KUKA KRL program: MyProgram_141().src

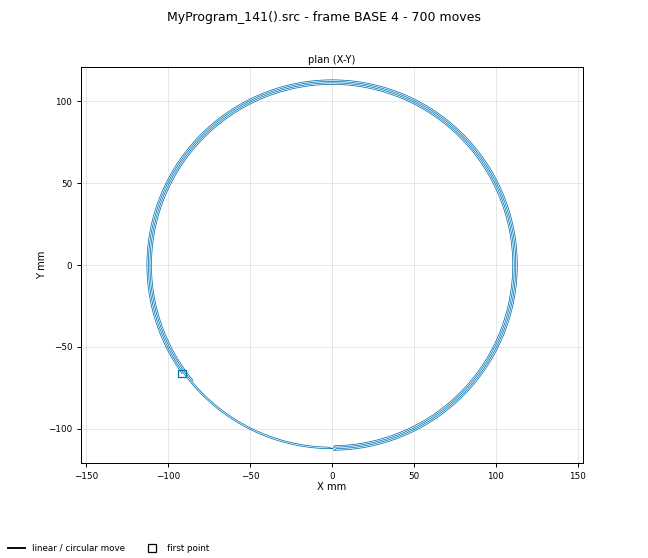
[picture p0: tool path of MyProgram_141().src in frame BASE 4, 700 of 700 moves have a stored position in this frame; points joined in program order, loops and branches not executed]
&ACCESS RVP
&REL 1
&PARAM TEMPLATE = C:\KRC\Roboter\Template\vorgabe
&PARAM EDITMASK = *
DEF MyProgram_141()
; ---- Setting reference (Base) ----
$BASE = BASE_DATA[4]

; --------------------------
; ---- Setting tool (TCP) ----
$TOOL = TOOL_DATA[3]
; --------------------------

$VEL.CP = VEL_APROX_PRINT
Startdeposition()
$VEL.CP = VEL_PRINT
LIN {X -91.6624,Y -66.2535,Z 113,A -148.3007,B 24.9515,C -1.6085,E1 24.8697,E2 234.2722} C_DIS
LIN {X -93.2607,Y -63.984,Z 113,A -149.7147,B 24.9513,C -1.6118,E1 24.8675,E2 235.6855} C_DIS
LIN {X -95.2768,Y -60.9377,Z 113,A -151.5758,B 24.9511,C -1.6162,E1 24.8646,E2 237.5454} C_DIS
LIN {X -96.7436,Y -58.5812,Z 113,A -152.9901,B 24.9508,C -1.6196,E1 24.8626,E2 238.9588} C_DIS
LIN {X -98.1521,Y -56.1893,Z 113,A -154.4681,B 24.9508,C -1.6206,E1 24.8605,E2 240.4422} C_DIS
LIN {X -99.7449,Y -53.3148,Z 113,A -156.2521,B 24.9508,C -1.6204,E1 24.8581,E2 242.2361} C_DIS
LIN {X -101.3464,Y -50.1991,Z 113,A -157.8945,B 24.9502,C -1.6306,E1 24.8561,E2 243.863} C_DIS
LIN {X -102.8265,Y -47.098,Z 113,A -159.6163,B 24.9498,C -1.6363,E1 24.854,E2 245.5806} C_DIS
LIN {X -103.9236,Y -44.624,Z 113,A -160.981,B 24.9496,C -1.6405,E1 24.8525,E2 246.9428} C_DIS
LIN {X -105.5211,Y -40.704,Z 113,A -163.1541,B 24.9493,C -1.6456,E1 24.8502,E2 249.1158} C_DIS
LIN {X -106.7787,Y -37.2743,Z 113,A -165.0805,B 24.9491,C -1.6482,E1 24.8484,E2 251.047} C_DIS
LIN {X -108.1071,Y -33.2262,Z 113,A -167.1751,B 24.9485,C -1.6572,E1 24.8466,E2 253.1321} C_DIS
LIN {X -108.8635,Y -30.6564,Z 113,A -168.6194,B 24.9485,C -1.658,E1 24.8455,E2 254.583} C_DIS
LIN {X -109.9181,Y -26.6287,Z 113,A -170.6791,B 24.948,C -1.6664,E1 24.8441,E2 256.6346} C_DIS
LIN {X -110.6473,Y -23.4242,Z 113,A -172.3554,B 24.9477,C -1.6711,E1 24.8431,E2 258.3095} C_DIS
LIN {X -111.3441,Y -19.8383,Z 113,A -174.2824,B 24.9475,C -1.674,E1 24.8421,E2 260.241} C_DIS
LIN {X -111.7974,Y -17.0998,Z 113,A -175.6982,B 24.9472,C -1.6781,E1 24.8415,E2 261.6556} C_DIS
LIN {X -112.3511,Y -12.9732,Z 113,A -177.8222,B 24.9468,C -1.6842,E1 24.8407,E2 263.7775} C_DIS
LIN {X -112.6356,Y -10.2121,Z 113,A -179.2383,B 24.9466,C -1.6884,E1 24.8403,E2 265.1923} C_DIS
LIN {X -112.8868,Y -6.9354,Z 113,A 179.149,B 24.9461,C -1.6957,E1 24.84,E2 266.7972} C_DIS
LIN {X -113.001,Y -4.673,Z 113,A 177.9295,B 24.9461,C -1.6967,E1 24.8399,E2 268.0217} C_DIS
LIN {X -113.097,Y -0.5539,Z 113,A 175.7974,B 24.9457,C -1.7017,E1 24.8398,E2 270.1548} C_DIS
LIN {X -113.0655,Y 2.7756,Z 113,A 174.1926,B 24.9452,C -1.7103,E1 24.8398,E2 271.7486} C_DIS
LIN {X -112.9676,Y 5.4512,Z 113,A 172.8457,B 24.9449,C -1.7151,E1 24.84,E2 273.0923} C_DIS
LIN {X -112.8276,Y 7.8107,Z 113,A 171.6206,B 24.9447,C -1.7179,E1 24.8402,E2 274.3179} C_DIS
LIN {X -112.555,Y 11.0857,Z 113,A 169.944,B 24.9444,C -1.7228,E1 24.8407,E2 275.9929} C_DIS
LIN {X -112.249,Y 13.8446,Z 113,A 168.5279,B 24.9441,C -1.727,E1 24.8411,E2 277.4075} C_DIS
LIN {X -111.9473,Y 16.0896,Z 113,A 167.3084,B 24.9441,C -1.728,E1 24.8416,E2 278.6319} C_DIS
LIN {X -111.4345,Y 19.3357,Z 113,A 165.6956,B 24.9436,C -1.7354,E1 24.8423,E2 280.2368} C_DIS
LIN {X -110.75,Y 22.924,Z 113,A 163.8317,B 24.9432,C -1.7408,E1 24.8433,E2 282.0987} C_DIS
LIN {X -110.0391,Y 26.1326,Z 113,A 162.1555,B 24.9429,C -1.7457,E1 24.8444,E2 283.7731} C_DIS
LIN {X -109.3647,Y 28.8252,Z 113,A 160.7396,B 24.9426,C -1.7498,E1 24.8453,E2 285.1874} C_DIS
LIN {X -108.3748,Y 32.3415,Z 113,A 158.8759,B 24.9423,C -1.7552,E1 24.8468,E2 287.0491} C_DIS
LIN {X -107.5485,Y 34.9914,Z 113,A 157.4602,B 24.942,C -1.7593,E1 24.848,E2 288.4632} C_DIS
LIN {X -106.4883,Y 38.1021,Z 113,A 155.7838,B 24.9417,C -1.764,E1 24.8495,E2 290.1378} C_DIS
LIN {X -105.2004,Y 41.5206,Z 113,A 153.857,B 24.9415,C -1.7668,E1 24.8514,E2 292.0687} C_DIS
LIN {X -103.6008,Y 45.3645,Z 113,A 151.7972,B 24.9409,C -1.7752,E1 24.8537,E2 294.12} C_DIS
LIN {X -102.2408,Y 48.3563,Z 113,A 150.1215,B 24.9406,C -1.7798,E1 24.8556,E2 295.794} C_DIS
LIN {X -100.6241,Y 51.6321,Z 113,A 148.1949,B 24.9405,C -1.7824,E1 24.8581,E2 297.7247} C_DIS
LIN {X -99.0832,Y 54.5348,Z 113,A 146.5831,B 24.94,C -1.7893,E1 24.8602,E2 299.3284} C_DIS
LIN {X -97.9694,Y 56.5073,Z 113,A 145.3647,B 24.94,C -1.7899,E1 24.8619,E2 300.5518} C_DIS
LIN {X -96.5531,Y 58.8945,Z 113,A 143.9497,B 24.9397,C -1.7936,E1 24.8639,E2 301.9652} C_DIS
LIN {X -94.8029,Y 61.676,Z 113,A 142.3381,B 24.9392,C -1.8004,E1 24.8663,E2 303.5688} C_DIS
LIN {X -92.4685,Y 65.1237,Z 113,A 140.2161,B 24.9389,C -1.8058,E1 24.8697,E2 305.6885} C_DIS
LIN {X -90.8425,Y 67.3734,Z 113,A 138.8015,B 24.9386,C -1.8093,E1 24.872,E2 307.1016} C_DIS
LIN {X -88.6177,Y 70.2707,Z 113,A 136.9398,B 24.9383,C -1.8139,E1 24.8752,E2 308.9611} C_DIS
LIN {X -86.5401,Y 72.8171,Z 113,A 135.2656,B 24.9381,C -1.8179,E1 24.8782,E2 310.6337} C_DIS
LIN {X -84.1419,Y 75.5726,Z 113,A 133.4046,B 24.9378,C -1.8222,E1 24.8816,E2 312.4926} C_DIS
LIN {X -81.9121,Y 77.9868,Z 113,A 131.7306,B 24.9375,C -1.826,E1 24.8848,E2 314.165} C_DIS
LIN {X -79.9735,Y 79.9735,Z 113,A 130.317,B 24.9373,C -1.8292,E1 24.8875,E2 315.5771} C_DIS
LIN {X -77.3477,Y 82.5131,Z 113,A 128.4565,B 24.937,C -1.8332,E1 24.8913,E2 317.4356} C_DIS
LIN {X -75.2994,Y 84.3864,Z 113,A 127.0431,B 24.9368,C -1.8362,E1 24.8942,E2 318.8476} C_DIS
LIN {X -73.2058,Y 86.209,Z 113,A 125.6303,B 24.9366,C -1.8391,E1 24.8972,E2 320.2589} C_DIS
LIN {X -71.0681,Y 87.9796,Z 113,A 124.217,B 24.9364,C -1.8419,E1 24.9003,E2 321.6708} C_DIS
LIN {X -68.4831,Y 90.0088,Z 113,A 122.5445,B 24.9362,C -1.8452,E1 24.9039,E2 323.3419} C_DIS
LIN {X -65.1237,Y 92.4685,Z 113,A 120.4259,B 24.9359,C -1.8491,E1 24.9087,E2 325.4583} C_DIS
LIN {X -62.1023,Y 94.5218,Z 113,A 118.5671,B 24.9357,C -1.8525,E1 24.913,E2 327.3154} C_DIS
LIN {X -59.764,Y 96.0174,Z 113,A 117.155,B 24.9355,C -1.8549,E1 24.9164,E2 328.7261} C_DIS
LIN {X -57.5917,Y 97.3357,Z 113,A 115.8128,B 24.9355,C -1.8551,E1 24.9196,E2 330.0721} C_DIS
LIN {X -55.0035,Y 98.8214,Z 113,A 114.2756,B 24.9354,C -1.8567,E1 24.9233,E2 331.6098} C_DIS
LIN {X -52.0867,Y 100.3917,Z 113,A 112.6607,B 24.935,C -1.8621,E1 24.9273,E2 333.2165} C_DIS
LIN {X -50.0648,Y 101.4129,Z 113,A 111.4638,B 24.935,C -1.862,E1 24.9303,E2 334.4168} C_DIS
LIN {X -47.098,Y 102.8265,Z 113,A 109.8386,B 24.9347,C -1.8661,E1 24.9344,E2 336.0362} C_DIS
LIN {X -44.5603,Y 103.9514,Z 113,A 108.4276,B 24.9346,C -1.868,E1 24.938,E2 337.4461} C_DIS
LIN {X -42.0475,Y 104.9926,Z 113,A 107.0448,B 24.9345,C -1.8698,E1 24.9416,E2 338.8278} C_DIS
LIN {X -39.406,Y 106.0127,Z 113,A 105.6067,B 24.9343,C -1.8715,E1 24.9453,E2 340.2648} C_DIS
LIN {X -35.83,Y 107.2723,Z 113,A 103.6446,B 24.9343,C -1.8723,E1 24.9505,E2 342.229} C_DIS
LIN {X -32.8311,Y 108.2296,Z 113,A 102.0821,B 24.9341,C -1.8754,E1 24.9547,E2 343.7867} C_DIS
LIN {X -28.8252,Y 109.3647,Z 113,A 99.968,B 24.9339,C -1.8774,E1 24.9604,E2 345.8993} C_DIS
LIN {X -25.2778,Y 110.2366,Z 113,A 98.0502,B 24.9339,C -1.8764,E1 24.9656,E2 347.822} C_DIS
LIN {X -22.5648,Y 110.8237,Z 113,A 96.6414,B 24.9339,C -1.8775,E1 24.9694,E2 349.2299} C_DIS
LIN {X -19.8383,Y 111.3441,Z 113,A 95.2326,B 24.9339,C -1.8785,E1 24.9733,E2 350.6378} C_DIS
LIN {X -17.0998,Y 111.7974,Z 113,A 93.8243,B 24.9338,C -1.8794,E1 24.9772,E2 352.0453} C_DIS
LIN {X -13.8446,Y 112.249,Z 113,A 92.2208,B 24.9335,C -1.883,E1 24.9816,E2 353.6416} C_DIS
LIN {X -11.0857,Y 112.555,Z 113,A 90.8126,B 24.9335,C -1.8836,E1 24.9855,E2 355.049} C_DIS
LIN {X -7.8107,Y 112.8276,Z 113,A 89.1098,B 24.9335,C -1.8828,E1 24.9902,E2 356.7544} C_DIS
LIN {X -4.673,Y 113.001,Z 113,A 87.4895,B 24.9335,C -1.8822,E1 24.9948,E2 358.3766} C_DIS
LIN {X -1.8984,Y 113.0817,Z 113,A 86.0825,B 24.9335,C -1.8825,E1 24.9987,E2 359.7829} C_DIS
LIN {X 0.8773,Y 113.0942,Z 113,A 84.6757,B 24.9335,C -1.8828,E1 25.0026,E2 361.189} C_DIS
LIN {X 3.6525,Y 113.0386,Z 113,A 83.2692,B 24.9335,C -1.8829,E1 25.0066,E2 362.595} C_DIS
LIN {X 7.8107,Y 112.8276,Z 113,A 81.1598,B 24.9335,C -1.8829,E1 25.0124,E2 364.7035} C_DIS
LIN {X 11.0857,Y 112.555,Z 113,A 79.5585,B 24.9334,C -1.8854,E1 25.0169,E2 366.2981} C_DIS
LIN {X 13.8446,Y 112.249,Z 113,A 78.1528,B 24.9334,C -1.8852,E1 25.0208,E2 367.7033} C_DIS
LIN {X 17.9668,Y 111.6634,Z 113,A 76.0447,B 24.9334,C -1.8846,E1 25.0266,E2 369.8107} C_DIS
LIN {X 20.7017,Y 111.1888,Z 113,A 74.6394,B 24.9334,C -1.8841,E1 25.0304,E2 371.2156} C_DIS
LIN {X 24.2814,Y 110.4603,Z 113,A 72.7275,B 24.9337,C -1.8807,E1 25.0357,E2 373.1332} C_DIS
LIN {X 28.3307,Y 109.4918,Z 113,A 70.6209,B 24.9337,C -1.8796,E1 25.0414,E2 375.2394} C_DIS
LIN {X 32.3415,Y 108.3748,Z 113,A 68.5776,B 24.9337,C -1.8809,E1 25.0469,E2 377.2761} C_DIS
LIN {X 35.4773,Y 107.3913,Z 113,A 66.9158,B 24.9337,C -1.8797,E1 25.0513,E2 378.9378} C_DIS
LIN {X 38.1021,Y 106.4883,Z 113,A 65.5124,B 24.9338,C -1.8785,E1 25.055,E2 380.3411} C_DIS
LIN {X 41.5206,Y 105.2004,Z 113,A 63.6021,B 24.9342,C -1.8742,E1 25.06,E2 382.2574} C_DIS
LIN {X 45.3646,Y 103.6008,Z 113,A 61.5608,B 24.9342,C -1.8749,E1 25.0652,E2 384.2924} C_DIS
LIN {X 47.8934,Y 102.4563,Z 113,A 60.1581,B 24.9342,C -1.8734,E1 25.0688,E2 385.695} C_DIS
LIN {X 50.4481,Y 101.223,Z 113,A 58.6745,B 24.9345,C -1.8695,E1 25.0725,E2 387.1838} C_DIS
LIN {X 53.3148,Y 99.7449,Z 113,A 57.0957,B 24.9345,C -1.8697,E1 25.0764,E2 388.7577} C_DIS
LIN {X 55.7466,Y 98.4065,Z 113,A 55.6935,B 24.9345,C -1.8679,E1 25.0798,E2 390.1601} C_DIS
LIN {X 58.8945,Y 96.5531,Z 113,A 53.8489,B 24.9348,C -1.8655,E1 25.0842,E2 392.0047} C_DIS
LIN {X 61.2463,Y 95.0787,Z 113,A 52.3843,B 24.9351,C -1.8607,E1 25.0877,E2 393.476} C_DIS
LIN {X 63.984,Y 93.2607,Z 113,A 50.7882,B 24.9351,C -1.8609,E1 25.0914,E2 395.0661} C_DIS
LIN {X 66.7663,Y 91.2869,Z 113,A 49.0153,B 24.9354,C -1.856,E1 25.0954,E2 396.8444} C_DIS
LIN {X 69.5825,Y 89.1617,Z 113,A 47.2861,B 24.9354,C -1.8553,E1 25.0992,E2 398.569} C_DIS
LIN {X 71.7496,Y 87.4272,Z 113,A 45.8855,B 24.9356,C -1.8529,E1 25.1023,E2 399.97} C_DIS
LIN {X 74.5344,Y 85.0629,Z 113,A 44.0427,B 24.9359,C -1.8496,E1 25.1062,E2 401.8133} C_DIS
LIN {X 76.9757,Y 82.8629,Z 113,A 42.385,B 24.9361,C -1.8465,E1 25.1096,E2 403.4716} C_DIS
LIN {X 78.782,Y 81.1456,Z 113,A 41.1061,B 24.9363,C -1.8432,E1 25.1122,E2 404.7532} C_DIS
LIN {X 80.9489,Y 78.9861,Z 113,A 39.5855,B 24.9365,C -1.8411,E1 25.1152,E2 406.2722} C_DIS
LIN {X 83.456,Y 76.3293,Z 113,A 37.7435,B 24.9367,C -1.8374,E1 25.1187,E2 408.1149} C_DIS
LIN {X 85.2305,Y 74.3424,Z 113,A 36.3792,B 24.937,C -1.8336,E1 25.1212,E2 409.4819} C_DIS
LIN {X 87.1008,Y 72.1424,Z 113,A 34.9452,B 24.9371,C -1.8315,E1 25.1238,E2 410.9144} C_DIS
LIN {X 88.8451,Y 69.9831,Z 113,A 33.4832,B 24.9375,C -1.8256,E1 25.1263,E2 412.3835} C_DIS
LIN {X 91.3607,Y 66.6655,Z 113,A 31.4479,B 24.9377,C -1.8237,E1 25.1297,E2 414.4136} C_DIS
LIN {X 92.9693,Y 64.4033,Z 113,A 29.9866,B 24.9381,C -1.8176,E1 25.1321,E2 415.8821} C_DIS
LIN {X 95.2768,Y 60.9377,Z 113,A 27.8889,B 24.9384,C -1.8127,E1 25.1353,E2 417.981} C_DIS
LIN {X 97.0088,Y 58.1448,Z 113,A 26.2963,B 24.9384,C -1.8114,E1 25.1376,E2 419.5683} C_DIS
LIN {X 98.8342,Y 54.9806,Z 113,A 24.4069,B 24.939,C -1.8047,E1 25.1402,E2 421.4638} C_DIS
LIN {X 100.1537,Y 52.5385,Z 113,A 22.9957,B 24.9392,C -1.8006,E1 25.1421,E2 422.8774} C_DIS
LIN {X 101.8609,Y 49.1471,Z 113,A 21.1008,B 24.9395,C -1.7964,E1 25.1444,E2 424.7718} C_DIS
LIN {X 103.187,Y 46.2982,Z 113,A 19.5015,B 24.9398,C -1.7915,E1 25.1463,E2 426.3741} C_DIS
LIN {X 104.4904,Y 43.2813,Z 113,A 17.91,B 24.9399,C -1.79,E1 25.148,E2 427.9605} C_DIS
LIN {X 106.0127,Y 39.406,Z 113,A 15.8138,B 24.9403,C -1.7844,E1 25.1501,E2 430.0583} C_DIS
LIN {X 107.2281,Y 35.9611,Z 113,A 13.9748,B 24.9407,C -1.7794,E1 25.1518,E2 431.8987} C_DIS
LIN {X 108.2296,Y 32.8311,Z 113,A 12.3208,B 24.941,C -1.7748,E1 25.1532,E2 433.5542} C_DIS
LIN {X 109.3647,Y 28.8252,Z 113,A 10.2255,B 24.9414,C -1.7689,E1 25.1548,E2 435.6513} C_DIS
LIN {X 110.0391,Y 26.1326,Z 113,A 8.8283,B 24.9416,C -1.765,E1 25.1557,E2 437.0497} C_DIS
LIN {X 110.6473,Y 23.4242,Z 113,A 7.4316,B 24.9419,C -1.761,E1 25.1565,E2 438.4476} C_DIS
LIN {X 111.3441,Y 19.8383,Z 113,A 5.5934,B 24.9422,C -1.7558,E1 25.1575,E2 440.2874} C_DIS
LIN {X 111.7974,Y 17.0998,Z 113,A 4.1339,B 24.9427,C -1.7489,E1 25.1581,E2 441.7546} C_DIS
LIN {X 112.249,Y 13.8446,Z 113,A 2.5434,B 24.9428,C -1.7469,E1 25.1587,E2 443.3403} C_DIS
LIN {X 112.555,Y 11.0857,Z 113,A 1.1463,B 24.9431,C -1.7428,E1 25.1591,E2 444.7387} C_DIS
LIN {X 112.8868,Y 6.9353,Z 113,A -0.9482,B 24.9435,C -1.7367,E1 25.1595,E2 446.8353} C_DIS
LIN {X 113.001,Y 4.673,Z 113,A -2.1507,B 24.9439,C -1.7305,E1 25.1597,E2 448.0453} C_DIS
LIN {X 113.097,Y 0.5539,Z 113,A -4.2532,B 24.9444,C -1.723,E1 25.1597,E2 450.1529} C_DIS
LIN {X 113.0655,Y -2.7756,Z 113,A -5.8358,B 24.9444,C -1.7223,E1 25.1597,E2 451.7278} C_DIS
LIN {X 112.9149,Y -6.4255,Z 113,A -7.6739,B 24.9448,C -1.7169,E1 25.1595,E2 453.5678} C_DIS
LIN {X 112.7232,Y -9.1946,Z 113,A -9.1329,B 24.9452,C -1.7099,E1 25.1592,E2 455.0346} C_DIS
LIN {X 112.4637,Y -11.9582,Z 113,A -10.5296,B 24.9455,C -1.7057,E1 25.1588,E2 456.4328} C_DIS
LIN {X 112.0707,Y -15.221,Z 113,A -12.12,B 24.9456,C -1.7037,E1 25.1582,E2 458.0186} C_DIS
LIN {X 111.6634,Y -17.9668,Z 113,A -13.5164,B 24.9459,C -1.6996,E1 25.1576,E2 459.4165} C_DIS
LIN {X 111.1888,Y -20.7017,Z 113,A -14.913,B 24.9461,C -1.6955,E1 25.1569,E2 460.8146} C_DIS
LIN {X 110.6473,Y -23.4242,Z 113,A -16.3098,B 24.9464,C -1.6914,E1 25.1561,E2 462.2129} C_DIS
LIN {X 109.7102,Y -27.481,Z 113,A -18.4043,B 24.9468,C -1.6853,E1 25.1548,E2 464.3097} C_DIS
LIN {X 108.6249,Y -31.4982,Z 113,A -20.498,B 24.9472,C -1.6792,E1 25.1532,E2 466.4057} C_DIS
LIN {X 107.5485,Y -34.9914,Z 113,A -22.3374,B 24.9475,C -1.674,E1 25.1517,E2 468.247} C_DIS
LIN {X 106.4883,Y -38.1021,Z 113,A -23.9911,B 24.9478,C -1.6692,E1 25.1502,E2 469.9026} C_DIS
LIN {X 105.2004,Y -41.5206,Z 113,A -25.8926,B 24.9483,C -1.6611,E1 25.1483,E2 471.8125} C_DIS
LIN {X 103.9514,Y -44.5603,Z 113,A -27.4836,B 24.9484,C -1.6594,E1 25.1466,E2 473.399} C_DIS
LIN {X 102.8265,Y -47.098,Z 113,A -28.8805,B 24.9486,C -1.6555,E1 25.1449,E2 474.7974} C_DIS
LIN {X 101.6397,Y -49.6073,Z 113,A -30.2777,B 24.9489,C -1.6516,E1 25.1433,E2 476.1961} C_DIS
LIN {X 100.6241,Y -51.6321,Z 113,A -31.4181,B 24.9491,C -1.6486,E1 25.1418,E2 477.3378} C_DIS
LIN {X 99.3267,Y -54.0859,Z 113,A -32.8155,B 24.9493,C -1.6448,E1 25.14,E2 478.7367} C_DIS
LIN {X 97.715,Y -56.95,Z 113,A -34.4698,B 24.9496,C -1.6403,E1 25.1377,E2 480.393} C_DIS
LIN {X 96.2879,Y -59.3309,Z 113,A -35.8672,B 24.9498,C -1.6367,E1 25.1356,E2 481.7918} C_DIS
LIN {X 94.8029,Y -61.676,Z 113,A -37.265,B 24.95,C -1.633,E1 25.1335,E2 483.1912} C_DIS
LIN {X 93.2607,Y -63.984,Z 113,A -38.663,B 24.9502,C -1.6295,E1 25.1313,E2 484.5907} C_DIS
LIN {X 91.1441,Y -66.9614,Z 113,A -40.5026,B 24.9505,C -1.6249,E1 25.1283,E2 486.4323} C_DIS
LIN {X 89.4733,Y -69.178,Z 113,A -41.9632,B 24.9509,C -1.6186,E1 25.1259,E2 487.9009} C_DIS
LIN {X 87.4272,Y -71.7496,Z 113,A -43.556,B 24.9509,C -1.6174,E1 25.1231,E2 489.489} C_DIS
LIN {X 85.64,Y -73.8736,Z 113,A -44.9545,B 24.9512,C -1.614,E1 25.1205,E2 490.889} C_DIS
LIN {X 83.2081,Y -76.5995,Z 113,A -46.7951,B 24.9514,C -1.6098,E1 25.1171,E2 492.7315} C_DIS
LIN {X 81.3032,Y -78.6184,Z 113,A -48.2563,B 24.9518,C -1.6037,E1 25.1143,E2 494.2007} C_DIS
LIN {X 79.3494,Y -80.59,Z 113,A -49.6553,B 24.952,C -1.6006,E1 25.1115,E2 495.601} C_DIS
LIN {X 76.9757,Y -82.8629,Z 113,A -51.2485,B 24.952,C -1.5998,E1 25.1083,E2 497.1896} C_DIS
LIN {X 74.919,Y -84.727,Z 113,A -52.6478,B 24.9522,C -1.5968,E1 25.1053,E2 498.5903} C_DIS
LIN {X 72.1424,Y -87.1008,Z 113,A -54.4897,B 24.9524,C -1.5931,E1 25.1014,E2 500.434} C_DIS
LIN {X 69.9831,Y -88.845,Z 113,A -55.952,B 24.9528,C -1.5874,E1 25.0982,E2 501.9041} C_DIS
LIN {X 67.3734,Y -90.8425,Z 113,A -57.5464,B 24.9528,C -1.587,E1 25.0947,E2 503.4938} C_DIS
LIN {X 65.1237,Y -92.4685,Z 113,A -58.9464,B 24.953,C -1.5844,E1 25.0915,E2 504.8952} C_DIS
LIN {X 62.1023,Y -94.5218,Z 113,A -60.7893,B 24.9532,C -1.581,E1 25.0872,E2 506.7397} C_DIS
LIN {X 59.764,Y -96.0174,Z 113,A -62.1897,B 24.9533,C -1.5786,E1 25.0839,E2 508.1414} C_DIS
LIN {X 57.3896,Y -97.4552,Z 113,A -63.5903,B 24.9534,C -1.5762,E1 25.0805,E2 509.5433} C_DIS
LIN {X 54.5348,Y -99.0832,Z 113,A -65.2489,B 24.9536,C -1.5735,E1 25.0765,E2 511.2035} C_DIS
LIN {X 52.0867,Y -100.3917,Z 113,A -66.6498,B 24.9537,C -1.5713,E1 25.073,E2 512.6056} C_DIS
LIN {X 48.8166,Y -102.0197,Z 113,A -68.557,B 24.9541,C -1.5658,E1 25.0682,E2 514.5208} C_DIS
LIN {X 46.2982,Y -103.187,Z 113,A -69.9586,B 24.9541,C -1.5638,E1 25.0647,E2 515.9235} C_DIS
LIN {X 42.4688,Y -104.8212,Z 113,A -72.0612,B 24.9543,C -1.561,E1 25.0592,E2 518.0278} C_DIS
LIN {X 39.406,Y -106.0127,Z 113,A -73.6585,B 24.9543,C -1.5617,E1 25.0551,E2 519.6201} C_DIS
LIN {X 35.4773,Y -107.3913,Z 113,A -75.7619,B 24.9544,C -1.5592,E1 25.0495,E2 521.7251} C_DIS
LIN {X 32.8311,Y -108.2296,Z 113,A -77.1646,B 24.9545,C -1.5577,E1 25.0458,E2 523.1288} C_DIS
LIN {X 28.8252,Y -109.3647,Z 113,A -79.269,B 24.9547,C -1.5556,E1 25.0401,E2 525.2348} C_DIS
LIN {X 25.2778,Y -110.2366,Z 113,A -81.1787,B 24.9549,C -1.5513,E1 25.0349,E2 527.1521} C_DIS
LIN {X 21.2032,Y -111.0923,Z 113,A -83.2213,B 24.9549,C -1.5523,E1 25.0293,E2 529.1896} C_DIS
LIN {X 17.9668,Y -111.6634,Z 113,A -84.8834,B 24.9549,C -1.5511,E1 25.0248,E2 530.8528} C_DIS
LIN {X 15.221,Y -112.0707,Z 113,A -86.2875,B 24.9549,C -1.5502,E1 25.0209,E2 532.2577} C_DIS
LIN {X 11.0857,Y -112.555,Z 113,A -88.3944,B 24.955,C -1.5491,E1 25.015,E2 534.3659} C_DIS
LIN {X 8.3201,Y -112.7932,Z 113,A -89.7987,B 24.955,C -1.5485,E1 25.0111,E2 535.7709} C_DIS
LIN {X 5.5495,Y -112.9634,Z 113,A -91.2041,B 24.9551,C -1.548,E1 25.0072,E2 537.1771} C_DIS
LIN {X 2.9206,Y -113.0611,Z 113,A -92.5119,B 24.9551,C -1.5486,E1 25.0035,E2 538.4831} C_DIS
LIN {X 0.7926,Y -113.0921,Z 113,A -93.1683,B 24.954,C -1.5666,E1 25.0018,E2 539.0966} C_DIS
Enddeposition()
LIN {X 0.7926,Y -113.0921,Z 113,A -93.1683,B 24.954,C -1.5666,E1 25.0018,E2 539.0966} C_DIS
Startdeposition()
$VEL.CP = VEL_PRINT
LIN {X 2.5112,Y -112.1455,Z 113,A -92.1451,B 24.9527,C -1.5891,E1 25.0049,E2 538.0202} C_DIS
LIN {X 8.5342,Y -111.8483,Z 113,A -89.0646,B 24.9527,C -1.5904,E1 25.0134,E2 534.938} C_DIS
LIN {X 11.7323,Y -111.5575,Z 113,A -87.3874,B 24.9525,C -1.5929,E1 25.0181,E2 533.2559} C_DIS
LIN {X 14.4396,Y -111.2394,Z 113,A -85.9602,B 24.9523,C -1.5953,E1 25.0221,E2 531.8241} C_DIS
LIN {X 17.4758,Y -110.8035,Z 113,A -84.3472,B 24.9521,C -1.5984,E1 25.0265,E2 530.2052} C_DIS
LIN {X 20.9501,Y -110.1992,Z 113,A -82.5997,B 24.9521,C -1.5975,E1 25.0313,E2 528.4617} C_DIS
LIN {X 23.9582,Y -109.5843,Z 113,A -81.0272,B 24.9521,C -1.5991,E1 25.0356,E2 526.8874} C_DIS
LIN {X 27.7429,Y -108.688,Z 113,A -78.9698,B 24.9518,C -1.6042,E1 25.0412,E2 524.821} C_DIS
LIN {X 31.8742,Y -107.5488,Z 113,A -76.8637,B 24.9518,C -1.603,E1 25.0469,E2 522.7212} C_DIS
LIN {X 35.1139,Y -106.5368,Z 113,A -75.0751,B 24.9516,C -1.6075,E1 25.0516,E2 520.9253} C_DIS
LIN {X 38.3768,Y -105.4037,Z 113,A -73.3742,B 24.9516,C -1.607,E1 25.0561,E2 519.229} C_DIS
LIN {X 41.5145,Y -104.2092,Z 113,A -71.46,B 24.9509,C -1.6183,E1 25.0611,E2 517.2924} C_DIS
LIN {X 44.6783,Y -102.8911,Z 113,A -69.8639,B 24.9512,C -1.614,E1 25.0652,E2 515.7103} C_DIS
LIN {X 49.5705,Y -100.6258,Z 113,A -67.1605,B 24.9511,C -1.6162,E1 25.072,E2 513.0087} C_DIS
LIN {X 52.3888,Y -99.1874,Z 113,A -65.6255,B 24.9511,C -1.6153,E1 25.0758,E2 511.4802} C_DIS
LIN {X 55.0783,Y -97.7204,Z 113,A -63.9299,B 24.9506,C -1.6239,E1 25.08,E2 509.7691} C_DIS
LIN {X 58.6737,Y -95.6052,Z 113,A -62.0003,B 24.9509,C -1.6189,E1 25.0846,E2 507.8574} C_DIS
LIN {X 61.0092,Y -94.132,Z 113,A -60.5316,B 24.9506,C -1.6242,E1 25.088,E2 506.3808} C_DIS
LIN {X 64.0536,Y -92.0861,Z 113,A -58.5905,B 24.9501,C -1.6311,E1 25.0925,E2 504.4301} C_DIS
LIN {X 67.1129,Y -89.8815,Z 113,A -56.7131,B 24.9501,C -1.6329,E1 25.0968,E2 502.555} C_DIS
LIN {X 70.2089,Y -87.4855,Z 113,A -54.8395,B 24.9501,C -1.6316,E1 25.1009,E2 500.6916} C_DIS
LIN {X 72.6167,Y -85.4959,Z 113,A -53.0723,B 24.9494,C -1.643,E1 25.1047,E2 498.9042} C_DIS
LIN {X 75.0079,Y -83.4061,Z 113,A -51.4123,B 24.9491,C -1.6485,E1 25.1082,E2 497.2379} C_DIS
LIN {X 77.8348,Y -80.7741,Z 113,A -49.55,B 24.9491,C -1.6482,E1 25.1119,E2 495.3839} C_DIS
LIN {X 80.4847,Y -78.1351,Z 113,A -47.5426,B 24.9485,C -1.6573,E1 25.1159,E2 493.3635} C_DIS
LIN {X 83.1854,Y -75.2546,Z 113,A -45.5747,B 24.9483,C -1.6602,E1 25.1196,E2 491.3975} C_DIS
LIN {X 85.5486,Y -72.5549,Z 113,A -43.7264,B 24.948,C -1.6658,E1 25.123,E2 489.5445} C_DIS
LIN {X 88.0435,Y -69.5058,Z 113,A -41.8472,B 24.948,C -1.665,E1 25.1262,E2 487.6757} C_DIS
LIN {X 89.9009,Y -67.087,Z 113,A -40.2598,B 24.9477,C -1.6706,E1 25.1289,E2 486.0826} C_DIS
LIN {X 91.8394,Y -64.4085,Z 113,A -38.4603,B 24.9471,C -1.6804,E1 25.1319,E2 484.2688} C_DIS
LIN {X 94.7779,Y -60.0021,Z 113,A -35.8423,B 24.9469,C -1.6841,E1 25.1359,E2 481.6553} C_DIS
LIN {X 96.7147,Y -56.8248,Z 113,A -34.0662,B 24.9469,C -1.6839,E1 25.1384,E2 479.8887} C_DIS
LIN {X 98.2445,Y -54.1399,Z 113,A -32.4123,B 24.9464,C -1.692,E1 25.1407,E2 478.2243} C_DIS
LIN {X 100.6478,Y -49.5261,Z 113,A -30.158,B 24.947,C -1.6814,E1 25.1435,E2 476.0068} C_DIS
LIN {X 101.7078,Y -47.31,Z 113,A -28.5242,B 24.9457,C -1.7027,E1 25.1455,E2 474.3319} C_DIS
LIN {X 103.5972,Y -43.0195,Z 113,A -26.2509,B 24.9456,C -1.7044,E1 25.148,E2 472.0669} C_DIS
LIN {X 104.7364,Y -40.1649,Z 113,A -24.5203,B 24.9448,C -1.7167,E1 25.1498,E2 470.3169} C_DIS
LIN {X 105.9424,Y -36.8647,Z 113,A -22.9043,B 24.9449,C -1.7141,E1 25.1513,E2 468.716} C_DIS
LIN {X 106.9636,Y -33.791,Z 113,A -21.167,B 24.9444,C -1.7231,E1 25.1528,E2 466.9673} C_DIS
LIN {X 107.9761,Y -30.3958,Z 113,A -19.4367,B 24.9442,C -1.7252,E1 25.1541,E2 465.2419} C_DIS
LIN {X 108.853,Y -27.0925,Z 113,A -17.7976,B 24.9442,C -1.7259,E1 25.1553,E2 463.6107} C_DIS
LIN {X 109.5657,Y -24.0433,Z 113,A -16.0317,B 24.9433,C -1.7387,E1 25.1564,E2 461.8248} C_DIS
LIN {X 110.3068,Y -20.3814,Z 113,A -14.1646,B 24.9431,C -1.743,E1 25.1574,E2 459.9586} C_DIS
LIN {X 110.8378,Y -17.254,Z 113,A -12.4625,B 24.9425,C -1.752,E1 25.1581,E2 458.2451} C_DIS
LIN {X 111.3567,Y -13.5133,Z 113,A -10.1714,B 24.9409,C -1.7751,E1 25.1589,E2 455.9132} C_DIS
LIN {X 111.7451,Y -9.7981,Z 113,A -8.8111,B 24.9422,C -1.7559,E1 25.1593,E2 454.6062} C_DIS
LIN {X 112.062,Y -4.9855,Z 113,A -6.6068,B 24.9425,C -1.752,E1 25.1597,E2 452.4243} C_DIS
LIN {X 112.1495,Y -2.2913,Z 113,A -4.9394,B 24.9413,C -1.7698,E1 25.1597,E2 450.7247} C_DIS
LIN {X 112.1668,Y 1.309,Z 113,A -2.9928,B 24.9406,C -1.7808,E1 25.1597,E2 448.7639} C_DIS
LIN {X 112.0632,Y 4.9571,Z 113,A -1.224,B 24.9405,C -1.7824,E1 25.1596,E2 447.0017} C_DIS
LIN {X 111.8321,Y 8.7368,Z 113,A 0.6673,B 24.9402,C -1.7867,E1 25.1592,E2 445.1116} C_DIS
LIN {X 111.5367,Y 11.9304,Z 113,A 2.2567,B 24.94,C -1.7897,E1 25.1588,E2 443.5245} C_DIS
LIN {X 111.0858,Y 15.5789,Z 113,A 4.1552,B 24.9395,C -1.7966,E1 25.1581,E2 441.6208} C_DIS
LIN {X 110.5476,Y 19.0322,Z 113,A 6.027,B 24.9388,C -1.8063,E1 25.1572,E2 439.7373} C_DIS
LIN {X 109.8105,Y 22.9015,Z 113,A 7.8832,B 24.9389,C -1.8054,E1 25.1562,E2 437.8938} C_DIS
LIN {X 109.027,Y 26.3793,Z 113,A 9.7018,B 24.9385,C -1.811,E1 25.1551,E2 436.0727} C_DIS
LIN {X 108.1044,Y 29.9431,Z 113,A 11.8899,B 24.9372,C -1.8309,E1 25.1534,E2 433.8501} C_DIS
LIN {X 106.752,Y 34.449,Z 113,A 14.0135,B 24.9375,C -1.8254,E1 25.1517,E2 431.7517} C_DIS
LIN {X 105.6578,Y 37.6756,Z 113,A 15.8302,B 24.9369,C -1.8341,E1 25.15,E2 429.9247} C_DIS
LIN {X 103.8793,Y 42.3298,Z 113,A 18.1635,B 24.9371,C -1.832,E1 25.1477,E2 427.6094} C_DIS
LIN {X 102.5513,Y 45.4579,Z 113,A 20.1472,B 24.936,C -1.8483,E1 25.1454,E2 425.598} C_DIS
LIN {X 101.1808,Y 48.4271,Z 113,A 21.6412,B 24.9362,C -1.845,E1 25.1436,E2 424.1198} C_DIS
LIN {X 99.6449,Y 51.5159,Z 113,A 23.4735,B 24.9356,C -1.8531,E1 25.1413,E2 422.2782} C_DIS
LIN {X 97.8767,Y 54.7985,Z 113,A 25.2621,B 24.9356,C -1.8531,E1 25.1389,E2 420.499} C_DIS
LIN {X 95.8357,Y 58.2943,Z 113,A 27.2678,B 24.9354,C -1.8558,E1 25.1361,E2 418.4971} C_DIS
LIN {X 94.1883,Y 60.9215,Z 113,A 28.9898,B 24.9347,C -1.8662,E1 25.1335,E2 416.7591} C_DIS
LIN {X 91.8164,Y 64.4416,Z 113,A 31.1083,B 24.9345,C -1.8695,E1 25.1301,E2 414.6433} C_DIS
LIN {X 89.8392,Y 67.1691,Z 113,A 33.2028,B 24.933,C -1.8908,E1 25.1266,E2 412.5087} C_DIS
LIN {X 87.6788,Y 69.9664,Z 113,A 34.4506,B 24.9345,C -1.8699,E1 25.1245,E2 411.316} C_DIS
LIN {X 86.2115,Y 71.7655,Z 113,A 35.7535,B 24.9339,C -1.878,E1 25.1222,E2 409.9999} C_DIS
LIN {X 84.3142,Y 73.9857,Z 113,A 38.4395,B 24.9298,C -1.9356,E1 25.117,E2 407.19} C_DIS
LIN {X 79.6225,Y 79.0129,Z 113,A 40.65,B 24.9334,C -1.8843,E1 25.1129,E2 405.11} C_DIS
LIN {X 77.1108,Y 81.4663,Z 113,A 42.5453,B 24.9328,C -1.8927,E1 25.1091,E2 403.203} C_DIS
LIN {X 74.6437,Y 83.7322,Z 113,A 44.2075,B 24.9328,C -1.894,E1 25.1056,E2 401.5444} C_DIS
LIN {X 72.224,Y 85.8305,Z 113,A 46.1022,B 24.9317,C -1.9086,E1 25.1015,E2 399.6224} C_DIS
LIN {X 69.3952,Y 88.1309,Z 113,A 47.7592,B 24.9321,C -1.903,E1 25.098,E2 397.9849} C_DIS
LIN {X 66.5837,Y 90.2744,Z 113,A 49.4846,B 24.9321,C -1.9027,E1 25.0941,E2 396.2665} C_DIS
LIN {X 63.8801,Y 92.2067,Z 113,A 51.1892,B 24.9319,C -1.9059,E1 25.0902,E2 394.5602} C_DIS
LIN {X 60.4321,Y 94.5025,Z 113,A 53.3724,B 24.9314,C -1.9122,E1 25.0851,E2 392.3691} C_DIS
LIN {X 56.9256,Y 96.6552,Z 113,A 55.4975,B 24.9311,C -1.9164,E1 25.08,E2 390.2407} C_DIS
LIN {X 53.5657,Y 98.5568,Z 113,A 57.419,B 24.9311,C -1.917,E1 25.0753,E2 388.3235} C_DIS
LIN {X 50.218,Y 100.3049,Z 113,A 59.3265,B 24.931,C -1.9185,E1 25.0706,E2 386.4176} C_DIS
LIN {X 47.1976,Y 101.7601,Z 113,A 60.9948,B 24.931,C -1.9187,E1 25.0664,E2 384.7533} C_DIS
LIN {X 44.5978,Y 102.9263,Z 113,A 62.4366,B 24.931,C -1.9197,E1 25.0627,E2 383.3125} C_DIS
LIN {X 39.7619,Y 104.889,Z 113,A 65.0881,B 24.9308,C -1.9218,E1 25.0558,E2 380.6621} C_DIS
LIN {X 36.9792,Y 105.9022,Z 113,A 66.5834,B 24.9308,C -1.9224,E1 25.0519,E2 379.1683} C_DIS
LIN {X 33.7832,Y 106.9661,Z 113,A 68.5526,B 24.9298,C -1.9345,E1 25.0466,E2 377.1741} C_DIS
LIN {X 28.9249,Y 108.3798,Z 113,A 70.8823,B 24.9305,C -1.9253,E1 25.0404,E2 374.8701} C_DIS
LIN {X 26.5374,Y 108.9884,Z 113,A 72.2083,B 24.9302,C -1.929,E1 25.0368,E2 373.5375} C_DIS
LIN {X 22.4898,Y 109.8951,Z 113,A 74.2886,B 24.9302,C -1.9284,E1 25.0311,E2 371.4612} C_DIS
LIN {X 18.8205,Y 110.583,Z 113,A 76.2275,B 24.9302,C -1.9304,E1 25.0258,E2 369.5196} C_DIS
LIN {X 15.4258,Y 111.1075,Z 113,A 78.0589,B 24.9299,C -1.9342,E1 25.0207,E2 367.6809} C_DIS
LIN {X 11.6901,Y 111.5619,Z 113,A 79.838,B 24.9303,C -1.9284,E1 25.0158,E2 365.9167} C_DIS
LIN {X 8.5342,Y 111.8483,Z 113,A 81.6027,B 24.9298,C -1.9347,E1 25.0109,E2 364.138} C_DIS
LIN {X 4.6784,Y 112.0752,Z 113,A 83.4431,B 24.9302,C -1.9291,E1 25.0058,E2 362.3116} C_DIS
LIN {X 0.9332,Y 112.1691,Z 113,A 85.4241,B 24.93,C -1.9316,E1 25.0002,E2 360.3249} C_DIS
LIN {X -2.5688,Y 112.1444,Z 113,A 87.0799,B 24.9305,C -1.9256,E1 24.9956,E2 358.6832} C_DIS
LIN {X -5.2848,Y 112.0491,Z 113,A 88.6698,B 24.9299,C -1.9336,E1 24.9911,E2 357.0741} C_DIS
LIN {X -9.527,Y 111.7689,Z 113,A 90.8489,B 24.9299,C -1.933,E1 24.9851,E2 354.8955} C_DIS
LIN {X -13.1388,Y 111.4006,Z 113,A 92.5474,B 24.9305,C -1.9255,E1 24.9804,E2 353.2138} C_DIS
LIN {X -16.3964,Y 110.9696,Z 113,A 94.4753,B 24.9298,C -1.9347,E1 24.975,E2 351.2623} C_DIS
LIN {X -20.6054,Y 110.2655,Z 113,A 96.5241,B 24.9303,C -1.9276,E1 24.9694,E2 349.2284} C_DIS
LIN {X -23.8315,Y 109.6119,Z 113,A 98.0937,B 24.9308,C -1.9216,E1 24.9652,E2 347.6712} C_DIS
LIN {X -26.9861,Y 108.879,Z 113,A 99.936,B 24.9303,C -1.9278,E1 24.9601,E2 345.8117} C_DIS
LIN {X -31.2506,Y 107.7338,Z 113,A 102.6543,B 24.9291,C -1.9445,E1 24.9527,E2 343.0494} C_DIS
LIN {X -35.2766,Y 106.483,Z 113,A 104.2874,B 24.9309,C -1.9204,E1 24.9485,E2 341.4704} C_DIS
LIN {X -38.5104,Y 105.3549,Z 113,A 105.9824,B 24.9312,C -1.916,E1 24.9441,E2 339.7825} C_DIS
LIN {X -43.4392,Y 103.4203,Z 113,A 108.3547,B 24.9324,C -1.8987,E1 24.938,E2 337.4461} C_DIS
LIN {X -47.0891,Y 101.8106,Z 113,A 110.7629,B 24.9316,C -1.9107,E1 24.9318,E2 335.0037} C_DIS
LIN {X -51.1534,Y 99.8301,Z 113,A 112.6323,B 24.9331,C -1.8892,E1 24.9272,E2 333.1805} C_DIS
LIN {X -54.4111,Y 98.0931,Z 113,A 115.0157,B 24.9319,C -1.906,E1 24.9213,E2 330.7504} C_DIS
LIN {X -57.967,Y 96.0347,Z 113,A 117.4555,B 24.9312,C -1.916,E1 24.9153,E2 328.2794} C_DIS
LIN {X -60.8822,Y 94.2135,Z 113,A 118.7279,B 24.9328,C -1.8931,E1 24.9124,E2 327.0574} C_DIS
LIN {X -63.4968,Y 92.4731,Z 113,A 120.4695,B 24.9327,C -1.8954,E1 24.9084,E2 325.3045} C_DIS
LIN {X -66.4364,Y 90.3823,Z 113,A 122.2479,B 24.9331,C -1.8891,E1 24.9044,E2 323.5349} C_DIS
LIN {X -69.5533,Y 88.006,Z 113,A 124.2045,B 24.9335,C -1.883,E1 24.9001,E2 321.5857} C_DIS
LIN {X -71.7345,Y 86.2373,Z 113,A 125.766,B 24.9334,C -1.8849,E1 24.8967,E2 320.0137} C_DIS
LIN {X -74.3359,Y 84.0075,Z 113,A 127.595,B 24.9334,C -1.884,E1 24.8928,E2 318.1796} C_DIS
LIN {X -77.2426,Y 81.3424,Z 113,A 129.6857,B 24.9336,C -1.8823,E1 24.8886,E2 316.0844} C_DIS
LIN {X -80.1311,Y 78.498,Z 113,A 131.6917,B 24.9341,C -1.8747,E1 24.8846,E2 314.0881} C_DIS
LIN {X -82.6374,Y 75.8536,Z 113,A 133.4468,B 24.9347,C -1.8658,E1 24.8813,E2 312.3464} C_DIS
LIN {X -85.1716,Y 72.9974,Z 113,A 135.589,B 24.9346,C -1.8684,E1 24.8774,E2 310.1884} C_DIS
LIN {X -89.245,Y 67.9592,Z 113,A 138.672,B 24.9358,C -1.8506,E1 24.8721,E2 307.1333} C_DIS
LIN {X -91.132,Y 65.4046,Z 113,A 140.4009,B 24.9358,C -1.8504,E1 24.8692,E2 305.3965} C_DIS
LIN {X -93.2596,Y 62.3362,Z 113,A 142.8955,B 24.9346,C -1.8683,E1 24.8652,E2 302.8468} C_DIS
LIN {X -95.5337,Y 58.7913,Z 113,A 144.3651,B 24.9369,C -1.8352,E1 24.8632,E2 301.4486} C_DIS
LIN {X -97.4592,Y 55.539,Z 113,A 146.427,B 24.9369,C -1.8348,E1 24.8602,E2 299.3771} C_DIS
LIN {X -99.2698,Y 52.2323,Z 113,A 148.3864,B 24.9372,C -1.8304,E1 24.8577,E2 297.4177} C_DIS
LIN {X -101.0156,Y 48.7709,Z 113,A 150.3696,B 24.9376,C -1.8246,E1 24.8552,E2 295.4376} C_DIS
LIN {X -102.4191,Y 45.7512,Z 113,A 152.1982,B 24.9376,C -1.8244,E1 24.8531,E2 293.5994} C_DIS
LIN {X -104.1692,Y 41.6159,Z 113,A 154.2678,B 24.9387,C -1.8086,E1 24.8509,E2 291.556} C_DIS
LIN {X -104.9992,Y 39.4709,Z 113,A 155.6301,B 24.9384,C -1.8123,E1 24.8495,E2 290.1773} C_DIS
LIN {X -106.1419,Y 36.2883,Z 113,A 158.023,B 24.937,C -1.8331,E1 24.8474,E2 287.7212} C_DIS
LIN {X -107.5997,Y 31.7026,Z 113,A 159.6337,B 24.9398,C -1.792,E1 24.8461,E2 286.1991} C_DIS
LIN {X -108.827,Y 27.1991,Z 113,A 162.0691,B 24.9402,C -1.7864,E1 24.8444,E2 283.763} C_DIS
LIN {X -109.5471,Y 24.1286,Z 113,A 163.7872,B 24.9402,C -1.7854,E1 24.8433,E2 282.0371} C_DIS
LIN {X -110.3529,Y 20.125,Z 113,A 165.6165,B 24.9414,C -1.7687,E1 24.8423,E2 280.2368} C_DIS
LIN {X -110.6972,Y 18.1374,Z 113,A 166.9357,B 24.9408,C -1.7766,E1 24.8417,E2 278.8909} C_DIS
LIN {X -111.2782,Y 14.1406,Z 113,A 168.949,B 24.9414,C -1.768,E1 24.8409,E2 276.8862} C_DIS
LIN {X -111.6561,Y 10.7624,Z 113,A 170.731,B 24.9417,C -1.7641,E1 24.8404,E2 275.1027} C_DIS
LIN {X -111.9636,Y 6.8803,Z 113,A 172.6769,B 24.9422,C -1.7559,E1 24.84,E2 273.1646} C_DIS
LIN {X -112.1101,Y 3.7604,Z 113,A 174.3004,B 24.9425,C -1.7519,E1 24.8398,E2 271.541} C_DIS
LIN {X -112.1725,Y 0.4893,Z 113,A 176.0039,B 24.9428,C -1.7477,E1 24.8398,E2 269.8371} C_DIS
LIN {X -112.1381,Y -2.8475,Z 113,A 177.7433,B 24.943,C -1.7436,E1 24.8398,E2 268.0972} C_DIS
LIN {X -112.0431,Y -5.4255,Z 113,A 179.1559,B 24.943,C -1.743,E1 24.8401,E2 266.6774} C_DIS
LIN {X -111.8272,Y -8.7986,Z 113,A -179.2143,B 24.9437,C -1.7337,E1 24.8404,E2 265.06} C_DIS
LIN {X -111.5594,Y -11.7139,Z 113,A -177.6566,B 24.9438,C -1.7314,E1 24.8408,E2 263.4986} C_DIS
LIN {X -111.1052,Y -15.4421,Z 113,A -175.818,B 24.9444,C -1.7221,E1 24.8415,E2 261.671} C_DIS
LIN {X -110.6796,Y -18.2428,Z 113,A -174.2032,B 24.9443,C -1.7241,E1 24.8422,E2 260.0419} C_DIS
LIN {X -109.9208,Y -22.3645,Z 113,A -172.061,B 24.9447,C -1.7174,E1 24.8433,E2 257.9029} C_DIS
LIN {X -108.8384,Y -27.1523,Z 113,A -169.5648,B 24.9453,C -1.7092,E1 24.8449,E2 255.4118} C_DIS
LIN {X -107.909,Y -30.6327,Z 113,A -167.553,B 24.9452,C -1.7103,E1 24.8464,E2 253.3855} C_DIS
LIN {X -106.6951,Y -34.6248,Z 113,A -165.6045,B 24.9461,C -1.6967,E1 24.848,E2 251.4585} C_DIS
LIN {X -105.4255,Y -38.3169,Z 113,A -163.6145,B 24.9464,C -1.6905,E1 24.8499,E2 249.4717} C_DIS
LIN {X -104.2608,Y -41.3831,Z 113,A -161.8046,B 24.9464,C -1.6909,E1 24.8517,E2 247.6507} C_DIS
LIN {X -102.7596,Y -44.9801,Z 113,A -159.3671,B 24.9457,C -1.703,E1 24.8545,E2 245.1711} C_DIS
LIN {X -101.0872,Y -48.6219,Z 113,A -157.8376,B 24.9473,C -1.6765,E1 24.8563,E2 243.6963} C_DIS
LIN {X -98.7944,Y -53.1276,Z 113,A -155.4572,B 24.9483,C -1.6613,E1 24.8593,E2 241.3394} C_DIS
LIN {X -96.9363,Y -56.4489,Z 113,A -153.2657,B 24.948,C -1.6659,E1 24.8623,E2 239.1256} C_DIS
LIN {X -94.6629,Y -60.182,Z 113,A -151.2176,B 24.9488,C -1.6526,E1 24.8653,E2 237.0986} C_DIS
LIN {X -92.2269,Y -63.851,Z 113,A -148.8292,B 24.9488,C -1.6524,E1 24.869,E2 234.6988} C_DIS
LIN {X -90.2863,Y -66.5675,Z 113,A -146.9132,B 24.9486,C -1.6566,E1 24.8722,E2 232.7636} C_DIS
LIN {X -87.9031,Y -69.6835,Z 113,A -145.0633,B 24.9493,C -1.6456,E1 24.8754,E2 230.9312} C_DIS
LIN {X -85.6854,Y -72.3943,Z 113,A -143.1854,B 24.9493,C -1.6449,E1 24.8787,E2 229.0462} C_DIS
LIN {X -83.1623,Y -75.2803,Z 113,A -141.2928,B 24.9497,C -1.6378,E1 24.8822,E2 227.162} C_DIS
LIN {X -80.5824,Y -78.0337,Z 113,A -139.3275,B 24.9499,C -1.6351,E1 24.886,E2 225.1946} C_DIS
LIN {X -77.7577,Y -80.8484,Z 113,A -137.236,B 24.95,C -1.6331,E1 24.8902,E2 223.0992} C_DIS
LIN {X -74.8316,Y -83.564,Z 113,A -135.2763,B 24.9505,C -1.6257,E1 24.8942,E2 221.1491} C_DIS
LIN {X -72.3613,Y -85.7135,Z 113,A -133.45,B 24.9503,C -1.6287,E1 24.8981,E2 219.3085} C_DIS
LIN {X -69.8926,Y -87.7378,Z 113,A -131.8976,B 24.9507,C -1.6225,E1 24.9015,E2 217.7651} C_DIS
LIN {X -67.1402,Y -89.8609,Z 113,A -130.081,B 24.9507,C -1.621,E1 24.9055,E2 215.9455} C_DIS
LIN {X -63.882,Y -92.2054,Z 113,A -128.154,B 24.9513,C -1.6125,E1 24.9099,E2 214.0322} C_DIS
LIN {X -61.292,Y -93.9484,Z 113,A -126.2727,B 24.9507,C -1.6218,E1 24.9144,E2 212.1227} C_DIS
LIN {X -57.2981,Y -96.435,Z 113,A -124.1045,B 24.9515,C -1.6085,E1 24.9195,E2 209.9794} C_DIS
LIN {X -54.4535,Y -98.0693,Z 113,A -122.3937,B 24.9515,C -1.6076,E1 24.9236,E2 208.2656} C_DIS
LIN {X -50.8369,Y -99.9919,Z 113,A -120.3101,B 24.9518,C -1.6045,E1 24.9288,E2 206.1836} C_DIS
LIN {X -46.9577,Y -101.8718,Z 113,A -118.1566,B 24.952,C -1.5999,E1 24.9342,E2 204.0357} C_DIS
LIN {X -42.4361,Y -103.836,Z 113,A -115.568,B 24.952,C -1.6002,E1 24.9409,E2 201.4404} C_DIS
LIN {X -39.4576,Y -105.0042,Z 113,A -113.9807,B 24.9522,C -1.5967,E1 24.945,E2 199.8581} C_DIS
LIN {X -36.1347,Y -106.1937,Z 113,A -112.0404,B 24.952,C -1.6009,E1 24.9502,E2 197.904} C_DIS
LIN {X -33.3975,Y -107.0857,Z 113,A -110.6458,B 24.9522,C -1.5966,E1 24.9539,E2 196.5171} C_DIS
LIN {X -29.7397,Y -108.1597,Z 113,A -108.6588,B 24.9522,C -1.597,E1 24.9592,E2 194.526} C_DIS
LIN {X -26.2672,Y -109.0544,Z 113,A -106.9307,B 24.9525,C -1.5916,E1 24.9639,E2 192.8084} C_DIS
LIN {X -22.9341,Y -109.8038,Z 113,A -105.1445,B 24.9525,C -1.5925,E1 24.9687,E2 191.0177} C_DIS
LIN {X -19.7953,Y -110.4122,Z 113,A -103.5223,B 24.9525,C -1.5914,E1 24.9732,E2 189.3963} C_DIS
LIN {X -16.0488,Y -111.019,Z 113,A -101.5105,B 24.9524,C -1.594,E1 24.9788,E2 187.3765} C_DIS
LIN {X -12.0677,Y -111.5224,Z 113,A -99.4351,B 24.9524,C -1.5948,E1 24.9845,E2 185.2979} C_DIS
LIN {X -8.3411,Y -111.8637,Z 113,A -97.0546,B 24.9511,C -1.615,E1 24.9913,E2 182.8686} C_DIS
LIN {X -4.3313,Y -112.0901,Z 113,A -95.6519,B 24.9528,C -1.5872,E1 24.995,E2 181.5316} C_DIS
LIN {X 0.796,Y -112.1393,Z 113,A -93.8798,B 24.9549,C -1.5519,E1 24.9999,E2 179.843} C_DIS
Enddeposition()
LIN {X 0.796,Y -112.1393,Z 113,A -93.8798,B 24.9549,C -1.5519,E1 24.9998,E2 179.843} C_DIS
Startdeposition()
$VEL.CP = VEL_PRINT
LIN {X -2.5976,Y -111.2189,Z 113,A -95.7064,B 24.9542,C -1.5641,E1 24.9947,E2 181.6408} C_DIS
LIN {X -7.5291,Y -110.9928,Z 113,A -98.0111,B 24.9536,C -1.5739,E1 24.9884,E2 183.9228} C_DIS
LIN {X -11.1953,Y -110.6838,Z 113,A -99.973,B 24.9537,C -1.5712,E1 24.9829,E2 185.8921} C_DIS
LIN {X -14.5846,Y -110.2881,Z 113,A -101.7933,B 24.9539,C -1.5689,E1 24.9778,E2 187.7192} C_DIS
LIN {X -18.217,Y -109.7463,Z 113,A -103.5745,B 24.9536,C -1.574,E1 24.9729,E2 189.4899} C_DIS
LIN {X -21.5581,Y -109.1404,Z 113,A -105.3728,B 24.9536,C -1.5726,E1 24.968,E2 191.2934} C_DIS
LIN {X -24.9365,Y -108.4171,Z 113,A -107.1,B 24.9535,C -1.5757,E1 24.9633,E2 193.0157} C_DIS
LIN {X -28.4586,Y -107.5478,Z 113,A -108.8608,B 24.9532,C -1.5811,E1 24.9586,E2 194.7659} C_DIS
LIN {X -31.3684,Y -106.7342,Z 113,A -110.4565,B 24.9532,C -1.5806,E1 24.9543,E2 196.3656} C_DIS
LIN {X -37.0194,Y -104.908,Z 113,A -113.4191,B 24.9528,C -1.5869,E1 24.9464,E2 199.3185} C_DIS
LIN {X -41.9165,Y -103.049,Z 113,A -116.4549,B 24.9535,C -1.5757,E1 24.9385,E2 202.3875} C_DIS
LIN {X -45.6515,Y -101.4497,Z 113,A -118.3715,B 24.9529,C -1.5851,E1 24.9336,E2 204.2862} C_DIS
LIN {X -48.6812,Y -100.0327,Z 113,A -120.5338,B 24.9539,C -1.5694,E1 24.928,E2 206.4914} C_DIS
LIN {X -51.6225,Y -98.5458,Z 113,A -121.856,B 24.9528,C -1.5867,E1 24.9249,E2 207.776} C_DIS
LIN {X -54.8935,Y -96.7635,Z 113,A -123.8371,B 24.9528,C -1.5868,E1 24.92,E2 209.7626} C_DIS
LIN {X -57.5139,Y -95.2278,Z 113,A -125.4939,B 24.9529,C -1.5854,E1 24.916,E2 211.4278} C_DIS
LIN {X -61.126,Y -92.9501,Z 113,A -127.5447,B 24.9523,C -1.5948,E1 24.9112,E2 213.463} C_DIS
LIN {X -65.8102,Y -89.6946,Z 113,A -130.4778,B 24.952,C -1.6,E1 24.9045,E2 216.3939} C_DIS
LIN {X -68.7091,Y -87.4945,Z 113,A -132.1364,B 24.9513,C -1.6119,E1 24.9009,E2 218.0301} C_DIS
LIN {X -71.6784,Y -85.0804,Z 113,A -134.4216,B 24.9518,C -1.6031,E1 24.8959,E2 220.345} C_DIS
LIN {X -74.3565,Y -82.7481,Z 113,A -136.2192,B 24.9516,C -1.608,E1 24.8922,E2 222.138} C_DIS
LIN {X -77.1468,Y -80.1528,Z 113,A -138.1844,B 24.9513,C -1.6119,E1 24.8882,E2 224.1019} C_DIS
LIN {X -79.8615,Y -77.449,Z 113,A -140.1563,B 24.9511,C -1.6162,E1 24.8843,E2 226.0719} C_DIS
LIN {X -82.2204,Y -74.9403,Z 113,A -141.9823,B 24.9509,C -1.6181,E1 24.8809,E2 227.9015} C_DIS
LIN {X -84.5734,Y -72.2735,Z 113,A -143.7314,B 24.9505,C -1.6256,E1 24.8777,E2 229.6407} C_DIS
LIN {X -86.585,Y -69.8513,Z 113,A -145.4753,B 24.9505,C -1.6246,E1 24.8746,E2 231.3949} C_DIS
LIN {X -90.34,Y -64.9224,Z 113,A -148.5645,B 24.9498,C -1.6365,E1 24.8694,E2 234.4709} C_DIS
LIN {X -92.4469,Y -61.8871,Z 113,A -151.1815,B 24.9512,C -1.6137,E1 24.8652,E2 237.1551} C_DIS
LIN {X -94.8561,Y -58.1256,Z 113,A -152.8094,B 24.9492,C -1.6457,E1 24.8629,E2 238.7151} C_DIS
LIN {X -96.4936,Y -55.3631,Z 113,A -154.4962,B 24.9491,C -1.6489,E1 24.8605,E2 240.403} C_DIS
LIN {X -97.8438,Y -52.9405,Z 113,A -156.0393,B 24.9491,C -1.6484,E1 24.8585,E2 241.9555} C_DIS
LIN {X -99.6529,Y -49.451,Z 113,A -157.6818,B 24.9478,C -1.6688,E1 24.8564,E2 243.5581} C_DIS
LIN {X -101.9183,Y -44.5956,Z 113,A -160.6535,B 24.9478,C -1.6684,E1 24.853,E2 246.547} C_DIS
LIN {X -103.2738,Y -41.3643,Z 113,A -162.682,B 24.948,C -1.665,E1 24.8508,E2 248.5949} C_DIS
LIN {X -104.6058,Y -37.8654,Z 113,A -164.5851,B 24.9476,C -1.6717,E1 24.8489,E2 250.4927} C_DIS
LIN {X -105.7857,Y -34.4312,Z 113,A -166.3293,B 24.947,C -1.6822,E1 24.8474,E2 252.222} C_DIS
LIN {X -106.5049,Y -32.1416,Z 113,A -168.2214,B 24.9483,C -1.6609,E1 24.8458,E2 254.1756} C_DIS
LIN {X -107.6371,Y -28.1167,Z 113,A -170.5734,B 24.9483,C -1.6601,E1 24.8442,E2 256.5434} C_DIS
LIN {X -108.7878,Y -23.2703,Z 113,A -172.4879,B 24.9463,C -1.6927,E1 24.843,E2 258.3914} C_DIS
LIN {X -109.4618,Y -19.8553,Z 113,A -174.1355,B 24.9456,C -1.7039,E1 24.8422,E2 260.022} C_DIS
LIN {X -110.1397,Y -15.6633,Z 113,A -176.5584,B 24.9457,C -1.7018,E1 24.8412,E2 262.4642} C_DIS
LIN {X -110.6551,Y -11.4695,Z 113,A -178.5504,B 24.9448,C -1.7158,E1 24.8405,E2 264.4348} C_DIS
LIN {X -110.953,Y -8.1186,Z 113,A 179.7337,B 24.9444,C -1.722,E1 24.8401,E2 266.1464} C_DIS
LIN {X -111.1533,Y -4.5907,Z 113,A 177.6367,B 24.9447,C -1.7173,E1 24.8399,E2 268.267} C_DIS
LIN {X -111.2491,Y -0.2197,Z 113,A 175.4744,B 24.944,C -1.728,E1 24.8398,E2 270.4169} C_DIS
LIN {X -111.2131,Y 2.8416,Z 113,A 173.7833,B 24.944,C -1.7288,E1 24.8398,E2 272.1164} C_DIS
LIN {X -111.0042,Y 7.3611,Z 113,A 171.3813,B 24.9437,C -1.7337,E1 24.8403,E2 274.5211} C_DIS
LIN {X -110.615,Y 11.8532,Z 113,A 169.2332,B 24.9427,C -1.7478,E1 24.8409,E2 276.6485} C_DIS
LIN {X -110.1584,Y 15.5318,Z 113,A 167.4455,B 24.942,C -1.7586,E1 24.8415,E2 278.4211} C_DIS
LIN {X -109.517,Y 19.5482,Z 113,A 164.6378,B 24.9434,C -1.7384,E1 24.8429,E2 281.2936} C_DIS
LIN {X -108.665,Y 23.8332,Z 113,A 163.2886,B 24.9406,C -1.7797,E1 24.8436,E2 282.5522} C_DIS
LIN {X -107.0225,Y 30.3689,Z 113,A 159.4913,B 24.9407,C -1.7783,E1 24.8462,E2 286.375} C_DIS
LIN {X -105.4786,Y 35.361,Z 113,A 156.8221,B 24.9401,C -1.7876,E1 24.8485,E2 289.0373} C_DIS
LIN {X -104.6492,Y 37.7466,Z 113,A 155.17,B 24.9407,C -1.7783,E1 24.8501,E2 290.7209} C_DIS
LIN {X -102.7936,Y 42.5439,Z 113,A 152.7803,B 24.9395,C -1.7963,E1 24.8525,E2 293.081} C_DIS
LIN {X -101.2255,Y 46.149,Z 113,A 150.6997,B 24.9392,C -1.8004,E1 24.8549,E2 295.1635} C_DIS
LIN {X -99.6517,Y 49.4535,Z 113,A 148.8382,B 24.9388,C -1.807,E1 24.8571,E2 297.0193} C_DIS
LIN {X -97.8616,Y 52.9077,Z 113,A 146.8623,B 24.9383,C -1.8139,E1 24.8597,E2 298.9891} C_DIS
LIN {X -95.9718,Y 56.2642,Z 113,A 144.8596,B 24.938,C -1.819,E1 24.8625,E2 300.9902} C_DIS
LIN {X -92.0359,Y 62.4941,Z 113,A 140.9698,B 24.9375,C -1.8261,E1 24.8684,E2 304.8826} C_DIS
LIN {X -89.5805,Y 65.9658,Z 113,A 138.2528,B 24.9385,C -1.812,E1 24.8729,E2 307.6464} C_DIS
LIN {X -86.9843,Y 69.3545,Z 113,A 135.9878,B 24.9382,C -1.8154,E1 24.8769,E2 309.9141} C_DIS
LIN {X -84.132,Y 72.7885,Z 113,A 134.2988,B 24.9362,C -1.8446,E1 24.8798,E2 311.541} C_DIS
LIN {X -82.0206,Y 75.158,Z 113,A 132.9006,B 24.9353,C -1.8579,E1 24.8824,E2 312.9138} C_DIS
LIN {X -78.8332,Y 78.496,Z 113,A 129.8805,B 24.9366,C -1.839,E1 24.8884,E2 315.992} C_DIS
LIN {X -76.393,Y 80.8719,Z 113,A 128.5619,B 24.9352,C -1.8599,E1 24.891,E2 317.2662} C_DIS
LIN {X -74.2528,Y 82.8409,Z 113,A 127.0061,B 24.9351,C -1.8612,E1 24.8942,E2 318.8252} C_DIS
LIN {X -71.635,Y 85.1174,Z 113,A 125.0637,B 24.9352,C -1.8591,E1 24.8983,E2 320.78} C_DIS
LIN {X -66.3092,Y 89.3285,Z 113,A 121.5945,B 24.9346,C -1.8677,E1 24.906,E2 324.2416} C_DIS
LIN {X -60.9475,Y 93.0678,Z 113,A 118.0479,B 24.9346,C -1.8674,E1 24.9142,E2 327.8008} C_DIS
LIN {X -56.893,Y 95.6001,Z 113,A 115.8241,B 24.9337,C -1.8813,E1 24.9194,E2 329.9984} C_DIS
LIN {X -53.7196,Y 97.42,Z 113,A 113.8483,B 24.9337,C -1.881,E1 24.9242,E2 331.9807} C_DIS
LIN {X -50.8478,Y 98.9478,Z 113,A 112.4172,B 24.9328,C -1.8934,E1 24.9277,E2 333.3861} C_DIS
LIN {X -47.9507,Y 100.3837,Z 113,A 110.5296,B 24.9332,C -1.8873,E1 24.9325,E2 335.2933} C_DIS
LIN {X -44.0766,Y 102.1446,Z 113,A 107.6859,B 24.9348,C -1.8649,E1 24.94,E2 338.197} C_DIS
LIN {X -39.6411,Y 103.9459,Z 113,A 105.9982,B 24.9324,C -1.8989,E1 24.9441,E2 339.8072} C_DIS
LIN {X -37.3688,Y 104.7854,Z 113,A 103.6823,B 24.9353,C -1.8583,E1 24.9505,E2 342.2244} C_DIS
LIN {X -31.718,Y 106.6305,Z 113,A 101.6748,B 24.9321,C -1.9035,E1 24.9556,E2 344.1278} C_DIS
LIN {X -26.5799,Y 108.0262,Z 113,A 98.8861,B 24.9321,C -1.9044,E1 24.9631,E2 346.9186} C_DIS
LIN {X -23.1887,Y 108.8056,Z 113,A 97.1071,B 24.9319,C -1.9065,E1 24.968,E2 348.6949} C_DIS
LIN {X -20.2458,Y 109.3916,Z 113,A 95.2156,B 24.9328,C -1.8938,E1 24.9732,E2 350.6185} C_DIS
LIN {X -15.668,Y 110.139,Z 113,A 93.2137,B 24.9315,C -1.9111,E1 24.9787,E2 352.5811} C_DIS
LIN {X -12.5555,Y 110.5378,Z 113,A 91.4438,B 24.9319,C -1.9058,E1 24.9836,E2 354.3648} C_DIS
LIN {X -8.8077,Y 110.8987,Z 113,A 89.575,B 24.9316,C -1.9096,E1 24.9888,E2 356.2255} C_DIS
LIN {X -5.0201,Y 111.1348,Z 113,A 87.6222,B 24.9316,C -1.9104,E1 24.9942,E2 358.177} C_DIS
LIN {X -1.536,Y 111.2385,Z 113,A 85.7285,B 24.9318,C -1.9068,E1 24.9995,E2 360.0794} C_DIS
LIN {X 2.0213,Y 111.2295,Z 113,A 84.0642,B 24.9313,C -1.914,E1 25.0041,E2 361.7264} C_DIS
LIN {X 5.0945,Y 111.1316,Z 113,A 82.4004,B 24.9315,C -1.9108,E1 25.0088,E2 363.3973} C_DIS
LIN {X 8.7483,Y 110.9034,Z 113,A 80.5345,B 24.9315,C -1.9116,E1 25.014,E2 365.2606} C_DIS
LIN {X 12.47,Y 110.5478,Z 113,A 78.5541,B 24.9317,C -1.909,E1 25.0195,E2 367.2457} C_DIS
LIN {X 15.9628,Y 110.0972,Z 113,A 76.7692,B 24.9317,C -1.9098,E1 25.0244,E2 369.0273} C_DIS
LIN {X 19.7332,Y 109.4838,Z 113,A 74.8177,B 24.9317,C -1.9098,E1 25.0298,E2 370.9768} C_DIS
LIN {X 23.4925,Y 108.7393,Z 113,A 72.8803,B 24.9316,C -1.9104,E1 25.0351,E2 372.9104} C_DIS
LIN {X 26.2223,Y 108.1134,Z 113,A 71.2716,B 24.9321,C -1.9026,E1 25.0395,E2 374.5352} C_DIS
LIN {X 30.2662,Y 107.0516,Z 113,A 68.7518,B 24.9333,C -1.8859,E1 25.0464,E2 377.0905} C_DIS
LIN {X 33.9838,Y 105.9305,Z 113,A 67.469,B 24.9313,C -1.9144,E1 25.0496,E2 378.3034} C_DIS
LIN {X 39.2512,Y 104.0935,Z 113,A 64.2815,B 24.9324,C -1.8985,E1 25.0581,E2 381.5221} C_DIS
LIN {X 43.1412,Y 102.5423,Z 113,A 62.2845,B 24.9321,C -1.903,E1 25.0632,E2 383.5038} C_DIS
LIN {X 48.0509,Y 100.3356,Z 113,A 59.5257,B 24.9323,C -1.9003,E1 25.0702,E2 386.2619} C_DIS
LIN {X 50.9653,Y 98.8877,Z 113,A 57.8236,B 24.9325,C -1.8971,E1 25.0744,E2 387.9672} C_DIS
LIN {X 54.1578,Y 97.1753,Z 113,A 55.615,B 24.9338,C -1.8799,E1 25.0799,E2 390.2101} C_DIS
LIN {X 58.655,Y 94.5293,Z 113,A 53.4255,B 24.9325,C -1.8972,E1 25.0851,E2 392.3519} C_DIS
LIN {X 62.3902,Y 92.1062,Z 113,A 50.9613,B 24.9333,C -1.8861,E1 25.0909,E2 394.8341} C_DIS
LIN {X 65.5487,Y 89.8861,Z 113,A 49.0556,B 24.9333,C -1.8862,E1 25.0952,E2 396.7328} C_DIS
LIN {X 67.581,Y 88.369,Z 113,A 47.6532,B 24.9338,C -1.8797,E1 25.0983,E2 398.1456} C_DIS
LIN {X 70.4662,Y 86.0863,Z 113,A 45.7214,B 24.9341,C -1.8745,E1 25.1025,E2 400.0824} C_DIS
LIN {X 73.246,Y 83.7325,Z 113,A 43.9644,B 24.9341,C -1.876,E1 25.1062,E2 401.8289} C_DIS
LIN {X 75.8588,Y 81.3743,Z 113,A 42.0499,B 24.9346,C -1.8679,E1 25.1102,E2 403.7549} C_DIS
LIN {X 78.6833,Y 78.6477,Z 113,A 40.2158,B 24.9343,C -1.8718,E1 25.1138,E2 405.5721} C_DIS
LIN {X 81.0033,Y 76.2533,Z 113,A 37.95,B 24.9363,C -1.8441,E1 25.1183,E2 407.8936} C_DIS
LIN {X 83.5237,Y 73.4851,Z 113,A 36.4723,B 24.9352,C -1.8593,E1 25.1209,E2 409.3287} C_DIS
LIN {X 86.0985,Y 70.4515,Z 113,A 34.3022,B 24.9359,C -1.8491,E1 25.1248,E2 411.5128} C_DIS
LIN {X 89.376,Y 66.2454,Z 113,A 31.6971,B 24.9359,C -1.8486,E1 25.1292,E2 414.1068} C_DIS
LIN {X 91.4294,Y 63.3781,Z 113,A 30.0287,B 24.9359,C -1.8506,E1 25.1319,E2 415.7624} C_DIS
LIN {X 93.2648,Y 60.6482,Z 113,A 28.1528,B 24.9367,C -1.8381,E1 25.1348,E2 417.6584} C_DIS
LIN {X 94.9781,Y 57.9248,Z 113,A 26.1324,B 24.9381,C -1.8177,E1 25.1378,E2 419.7166} C_DIS
LIN {X 96.8655,Y 54.7125,Z 113,A 24.6313,B 24.9372,C -1.8309,E1 25.1399,E2 421.1788} C_DIS
LIN {X 98.5253,Y 51.6615,Z 113,A 22.927,B 24.9372,C -1.8297,E1 25.1421,E2 422.8769} C_DIS
LIN {X 100.0319,Y 48.683,Z 113,A 20.9459,B 24.9384,C -1.8132,E1 25.1446,E2 424.8864} C_DIS
LIN {X 101.8813,Y 44.6806,Z 113,A 18.8985,B 24.9381,C -1.8166,E1 25.1469,E2 426.9145} C_DIS
LIN {X 103.0756,Y 41.8512,Z 113,A 16.3816,B 24.9412,C -1.7706,E1 25.1496,E2 429.5261} C_DIS
LIN {X 105.177,Y 36.253,Z 113,A 14.3625,B 24.9387,C -1.8084,E1 25.1514,E2 431.4448} C_DIS
LIN {X 107.1975,Y 29.7515,Z 113,A 10.6431,B 24.9401,C -1.7881,E1 25.1544,E2 435.1908} C_DIS
LIN {X 108.2904,Y 25.4853,Z 113,A 8.5451,B 24.9401,C -1.7887,E1 25.1558,E2 437.2752} C_DIS
LIN {X 108.9966,Y 22.2674,Z 113,A 6.8955,B 24.9402,C -1.7856,E1 25.1568,E2 438.9228} C_DIS
LIN {X 109.6877,Y 18.5675,Z 113,A 4.9314,B 24.9407,C -1.7783,E1 25.1578,E2 440.8924} C_DIS
LIN {X 110.2692,Y 14.7304,Z 113,A 2.9402,B 24.9411,C -1.7722,E1 25.1585,E2 442.8861} C_DIS
LIN {X 110.6404,Y 11.6106,Z 113,A 1.3724,B 24.9413,C -1.7693,E1 25.159,E2 444.4516} C_DIS
LIN {X 110.9715,Y 7.8441,Z 113,A -0.5993,B 24.9418,C -1.762,E1 25.1595,E2 446.429} C_DIS
LIN {X 111.163,Y 4.3646,Z 113,A -2.4571,B 24.9424,C -1.7533,E1 25.1597,E2 448.296} C_DIS
LIN {X 111.2481,Y 0.4187,Z 113,A -4.4738,B 24.9428,C -1.7474,E1 25.1597,E2 450.3147} C_DIS
LIN {X 111.1979,Y -3.3372,Z 113,A -6.2921,B 24.9428,C -1.7464,E1 25.1597,E2 452.1245} C_DIS
LIN {X 111.0921,Y -5.8907,Z 113,A -7.6105,B 24.9431,C -1.742,E1 25.1595,E2 453.4455} C_DIS
LIN {X 110.8697,Y -9.171,Z 113,A -9.2266,B 24.9433,C -1.74,E1 25.1592,E2 455.0568} C_DIS
LIN {X 110.5152,Y -12.7485,Z 113,A -11.1129,B 24.9438,C -1.7324,E1 25.1586,E2 456.9498} C_DIS
LIN {X 110.1556,Y -15.5517,Z 113,A -12.9166,B 24.9451,C -1.712,E1 25.1579,E2 458.7909} C_DIS
LIN {X 109.6521,Y -18.7804,Z 113,A -14.2706,B 24.9445,C -1.7213,E1 25.1573,E2 460.115} C_DIS
LIN {X 108.9746,Y -22.3749,Z 113,A -16.1046,B 24.9447,C -1.7175,E1 25.1563,E2 461.9473} C_DIS
LIN {X 108.118,Y -26.2034,Z 113,A -18.3358,B 24.9457,C -1.7015,E1 25.1549,E2 464.2033} C_DIS
LIN {X 107.0888,Y -30.1351,Z 113,A -20.7034,B 24.9469,C -1.6825,E1 25.1531,E2 466.602} C_DIS
LIN {X 105.9611,Y -33.8892,Z 113,A -22.2385,B 24.946,C -1.6978,E1 25.1518,E2 468.0924} C_DIS
LIN {X 104.8225,Y -37.2631,Z 113,A -24.0691,B 24.9463,C -1.6922,E1 25.1502,E2 469.926} C_DIS
LIN {X 103.8129,Y -39.9923,Z 113,A -26.2402,B 24.9485,C -1.6574,E1 25.1479,E2 472.1669} C_DIS
LIN {X 102.0052,Y -44.3963,Z 113,A -27.9158,B 24.9468,C -1.6846,E1 25.1461,E2 473.7693} C_DIS
LIN {X 100.5647,Y -47.574,Z 113,A -29.7334,B 24.9472,C -1.6782,E1 25.144,E2 475.5921} C_DIS
LIN {X 96.6634,Y -55.0678,Z 113,A -34.6055,B 24.9495,C -1.642,E1 25.1375,E2 480.5241} C_DIS
LIN {X 94.6056,Y -58.531,Z 113,A -36.4848,B 24.9493,C -1.6447,E1 25.1348,E2 482.3873} C_DIS
LIN {X 92.8352,Y -61.3003,Z 113,A -38.1146,B 24.9494,C -1.6427,E1 25.1323,E2 484.0137} C_DIS
LIN {X 89.9684,Y -65.4363,Z 113,A -40.3781,B 24.949,C -1.6502,E1 25.1287,E2 486.2487} C_DIS
LIN {X 87.7767,Y -68.3495,Z 113,A -42.1316,B 24.949,C -1.6506,E1 25.1257,E2 487.9928} C_DIS
LIN {X 85.0238,Y -71.7449,Z 113,A -44.546,B 24.9498,C -1.6373,E1 25.1214,E2 490.4274} C_DIS
LIN {X 82.8021,Y -74.2962,Z 113,A -46.2077,B 24.9498,C -1.6364,E1 25.1183,E2 492.0838} C_DIS
LIN {X 80.1666,Y -77.1325,Z 113,A -48.2029,B 24.9501,C -1.6314,E1 25.1145,E2 494.0822} C_DIS
LIN {X 77.4903,Y -79.8217,Z 113,A -50.1785,B 24.9505,C -1.6256,E1 25.1106,E2 496.0631} C_DIS
LIN {X 75.017,Y -82.15,Z 113,A -51.9008,B 24.9507,C -1.6227,E1 25.107,E2 497.7853} C_DIS
LIN {X 72.4164,Y -84.4517,Z 113,A -53.6904,B 24.9509,C -1.6185,E1 25.1033,E2 499.5777} C_DIS
LIN {X 70.4373,Y -86.11,Z 113,A -55.558,B 24.9525,C -1.5918,E1 25.0991,E2 501.5012} C_DIS
LIN {X 67.1762,Y -88.6773,Z 113,A -57.1652,B 24.9514,C -1.6105,E1 25.0956,E2 503.0584} C_DIS
LIN {X 64.0926,Y -90.932,Z 113,A -59.1689,B 24.9517,C -1.6048,E1 25.0911,E2 505.0687} C_DIS
LIN {X 61.0489,Y -93.0009,Z 113,A -60.7691,B 24.9512,C -1.614,E1 25.0874,E2 506.6416} C_DIS
LIN {X 58.7668,Y -94.4595,Z 113,A -62.9078,B 24.9533,C -1.5788,E1 25.0822,E2 508.8568} C_DIS
LIN {X 55.241,Y -96.5638,Z 113,A -64.5223,B 24.9522,C -1.5967,E1 25.0784,E2 510.424} C_DIS
LIN {X 52.8763,Y -97.8786,Z 113,A -66.3637,B 24.9535,C -1.5748,E1 25.0738,E2 512.312} C_DIS
LIN {X 49.3868,Y -99.6847,Z 113,A -68.1506,B 24.9531,C -1.5817,E1 25.0693,E2 514.0778} C_DIS
LIN {X 44.7963,Y -101.8309,Z 113,A -70.2481,B 24.952,C -1.5999,E1 25.0641,E2 516.127} C_DIS
LIN {X 39.4291,Y -104.0261,Z 113,A -73.438,B 24.9528,C -1.5868,E1 25.0558,E2 519.3407} C_DIS
LIN {X 35.8633,Y -105.3092,Z 113,A -75.4101,B 24.953,C -1.5833,E1 25.0506,E2 521.3169} C_DIS
LIN {X 32.6159,Y -106.3599,Z 113,A -76.9866,B 24.9527,C -1.5891,E1 25.0465,E2 522.8769} C_DIS
LIN {X 28.3115,Y -107.587,Z 113,A -79.3376,B 24.953,C -1.5845,E1 25.0401,E2 525.2348} C_DIS
LIN {X 24.8978,Y -108.4261,Z 113,A -81.2353,B 24.9533,C -1.579,E1 25.0349,E2 527.1428} C_DIS
LIN {X 21.1985,Y -109.2096,Z 113,A -83.1687,B 24.9533,C -1.5779,E1 25.0296,E2 529.0764} C_DIS
LIN {X 18.0079,Y -109.7813,Z 113,A -84.9225,B 24.9536,C -1.573,E1 25.0248,E2 530.84} C_DIS
LIN {X 14.3612,Y -110.3171,Z 113,A -86.7122,B 24.9534,C -1.5764,E1 25.0199,E2 532.6203} C_DIS
LIN {X 11.1173,Y -110.692,Z 113,A -88.4437,B 24.9536,C -1.5733,E1 25.015,E2 534.3579} C_DIS
LIN {X 8.7483,Y -110.9034,Z 113,A -89.8429,B 24.9541,C -1.5653,E1 25.0111,E2 535.7752} C_DIS
LIN {X 3.8265,Y -111.1828,Z 113,A -92.2109,B 24.9537,C -1.5715,E1 25.0045,E2 538.1277} C_DIS
LIN {X 0.7977,Y -111.2251,Z 113,A -93.8194,B 24.9539,C -1.5694,E1 25.0001,E2 539.741} C_DIS
Enddeposition()
LIN {X 0.7977,Y -111.2251,Z 113,A -93.8194,B 24.9539,C -1.5694,E1 25.0001,E2 539.741} C_DIS
Startdeposition()
$VEL.CP = VEL_PRINT
LIN {X 1.5292,Y -110.3136,Z 113,A -92.549,B 24.9506,C -1.6229,E1 25.004,E2 538.344} C_DIS
LIN {X 5.3956,Y -110.1931,Z 113,A -90.1295,B 24.9495,C -1.6412,E1 25.0108,E2 535.882} C_DIS
LIN {X 8.9419,Y -109.9602,Z 113,A -88.8479,B 24.9509,C -1.618,E1 25.0142,E2 534.656} C_DIS
LIN {X 12.0541,Y -109.6641,Z 113,A -87.0402,B 24.9504,C -1.6267,E1 25.0193,E2 532.8288} C_DIS
LIN {X 15.4516,Y -109.2357,Z 113,A -85.362,B 24.9506,C -1.6236,E1 25.0239,E2 531.1593} C_DIS
LIN {X 19.2525,Y -108.6306,Z 113,A -83.3329,B 24.9504,C -1.6264,E1 25.0295,E2 529.1255} C_DIS
LIN {X 22.8496,Y -107.933,Z 113,A -81.3656,B 24.9502,C -1.6309,E1 25.0349,E2 527.1503} C_DIS
LIN {X 27.6827,Y -106.7938,Z 113,A -79.2284,B 24.9512,C -1.6144,E1 25.0406,E2 525.0551} C_DIS
LIN {X 33.7346,Y -105.0392,Z 113,A -75.9062,B 24.9508,C -1.6201,E1 25.0496,E2 521.7249} C_DIS
LIN {X 37.2119,Y -103.8598,Z 113,A -72.4301,B 24.9464,C -1.6915,E1 25.0591,E2 518.0872} C_DIS
LIN {X 43.8401,Y -101.2388,Z 113,A -70.1761,B 24.95,C -1.633,E1 25.0645,E2 515.9769} C_DIS
LIN {X 46.7308,Y -99.9373,Z 113,A -68.3881,B 24.9495,C -1.6418,E1 25.0691,E2 514.1727} C_DIS
LIN {X 53.8454,Y -96.2905,Z 113,A -64.4318,B 24.9495,C -1.6401,E1 25.0789,E2 510.2312} C_DIS
LIN {X 56.204,Y -94.9331,Z 113,A -62.5249,B 24.9481,C -1.6645,E1 25.0836,E2 508.2724} C_DIS
LIN {X 61.1837,Y -91.8043,Z 113,A -60.024,B 24.9492,C -1.646,E1 25.0893,E2 505.8235} C_DIS
LIN {X 64.2515,Y -89.6827,Z 113,A -57.8131,B 24.9482,C -1.6621,E1 25.0945,E2 503.5822} C_DIS
LIN {X 70.6684,Y -84.7184,Z 113,A -53.7699,B 24.9482,C -1.6636,E1 25.1033,E2 499.5503} C_DIS
LIN {X 73.1253,Y -82.6091,Z 113,A -51.9447,B 24.9475,C -1.6739,E1 25.1072,E2 497.7082} C_DIS
LIN {X 75.7969,Y -80.163,Z 113,A -50.0792,B 24.9473,C -1.6777,E1 25.111,E2 495.8413} C_DIS
LIN {X 78.4404,Y -77.5777,Z 113,A -48.2343,B 24.9472,C -1.679,E1 25.1146,E2 494.001} C_DIS
LIN {X 80.9594,Y -74.9466,Z 113,A -46.2969,B 24.9467,C -1.6858,E1 25.1184,E2 492.056} C_DIS
LIN {X 83.2246,Y -72.4216,Z 113,A -44.608,B 24.9467,C -1.6871,E1 25.1215,E2 490.3716} C_DIS
LIN {X 87.6,Y -67.0637,Z 113,A -41.1593,B 24.9465,C -1.6902,E1 25.1275,E2 486.9316} C_DIS
LIN {X 89.0674,Y -65.1014,Z 113,A -39.7649,B 24.9459,C -1.6992,E1 25.1298,E2 485.5228} C_DIS
LIN {X 92.6197,Y -59.9412,Z 113,A -36.2215,B 24.9445,C -1.7214,E1 25.1354,E2 481.9445} C_DIS
LIN {X 95.71,Y -54.8706,Z 113,A -33.4545,B 24.9448,C -1.716,E1 25.1393,E2 479.2044} C_DIS
LIN {X 99.0873,Y -48.5097,Z 113,A -29.9161,B 24.9447,C -1.718,E1 25.1439,E2 475.68} C_DIS
LIN {X 100.7818,Y -44.8826,Z 113,A -27.7492,B 24.944,C -1.7283,E1 25.1464,E2 473.5006} C_DIS
LIN {X 102.734,Y -40.2112,Z 113,A -24.5673,B 24.9418,C -1.7615,E1 25.1498,E2 470.2579} C_DIS
LIN {X 104.0493,Y -36.6736,Z 113,A -23.342,B 24.9436,C -1.7343,E1 25.1509,E2 469.1037} C_DIS
LIN {X 106.2014,Y -29.8745,Z 113,A -19.7324,B 24.9432,C -1.7416,E1 25.154,E2 465.4973} C_DIS
LIN {X 107.3812,Y -25.3122,Z 113,A -16.9434,B 24.9416,C -1.7649,E1 25.1559,E2 462.6696} C_DIS
LIN {X 108.1304,Y -21.8884,Z 113,A -15.1174,B 24.9412,C -1.771,E1 25.1569,E2 460.8397} C_DIS
LIN {X 109.2597,Y -15.2827,Z 113,A -11.8179,B 24.941,C -1.774,E1 25.1584,E2 457.5525} C_DIS
LIN {X 109.6483,Y -12.2005,Z 113,A -9.8265,B 24.9395,C -1.7964,E1 25.159,E2 455.52} C_DIS
LIN {X 110.1096,Y -6.8823,Z 113,A -7.5176,B 24.9403,C -1.7844,E1 25.1595,E2 453.2532} C_DIS
LIN {X 110.278,Y -3.1632,Z 113,A -5.4485,B 24.9395,C -1.7969,E1 25.1598,E2 451.167} C_DIS
LIN {X 110.322,Y 0.628,Z 113,A -3.453,B 24.939,C -1.8044,E1 25.1598,E2 449.1656} C_DIS
LIN {X 110.2252,Y 4.6484,Z 113,A -1.4037,B 24.9386,C -1.8094,E1 25.1596,E2 447.1167} C_DIS
LIN {X 110.0094,Y 8.3263,Z 113,A 0.5404,B 24.9381,C -1.817,E1 25.1592,E2 445.1663} C_DIS
LIN {X 109.683,Y 11.8731,Z 113,A 2.4098,B 24.9377,C -1.8238,E1 25.1587,E2 443.2919} C_DIS
LIN {X 109.2169,Y 15.5841,Z 113,A 4.1975,B 24.9377,C -1.823,E1 25.158,E2 441.5166} C_DIS
LIN {X 108.6625,Y 19.0751,Z 113,A 6.1027,B 24.9371,C -1.832,E1 25.1571,E2 439.6015} C_DIS
LIN {X 108.0322,Y 22.3664,Z 113,A 7.6994,B 24.9371,C -1.831,E1 25.1563,E2 438.0164} C_DIS
LIN {X 107.416,Y 25.1616,Z 113,A 9.2377,B 24.9367,C -1.8379,E1 25.1553,E2 436.4706} C_DIS
LIN {X 106.3078,Y 29.499,Z 113,A 12.2124,B 24.9341,C -1.8745,E1 25.1531,E2 433.4268} C_DIS
LIN {X 105.0637,Y 33.6586,Z 113,A 13.7043,B 24.9361,C -1.8468,E1 25.1519,E2 432.0086} C_DIS
LIN {X 104.2037,Y 36.2335,Z 113,A 16.1406,B 24.9325,C -1.8975,E1 25.1496,E2 429.4665} C_DIS
LIN {X 102.2268,Y 41.4836,Z 113,A 18.146,B 24.9348,C -1.8649,E1 25.1476,E2 427.549} C_DIS
LIN {X 100.8604,Y 44.7083,Z 113,A 20.0546,B 24.9342,C -1.8742,E1 25.1454,E2 425.629} C_DIS
LIN {X 98.3759,Y 49.9347,Z 113,A 22.6547,B 24.9348,C -1.8646,E1 25.1423,E2 423.0655} C_DIS
LIN {X 97.0842,Y 52.4013,Z 113,A 25.2177,B 24.931,C -1.9187,E1 25.1388,E2 420.3883} C_DIS
LIN {X 94.4008,Y 57.094,Z 113,A 27.0584,B 24.9335,C -1.8828,E1 25.1363,E2 418.6416} C_DIS
LIN {X 92.8179,Y 59.6324,Z 113,A 28.6944,B 24.933,C -1.8906,E1 25.1338,E2 416.9956} C_DIS
LIN {X 90.4869,Y 63.1136,Z 113,A 30.7597,B 24.933,C -1.8913,E1 25.1306,E2 414.939} C_DIS
LIN {X 88.6428,Y 65.6814,Z 113,A 32.5919,B 24.9321,C -1.9038,E1 25.1275,E2 413.086} C_DIS
LIN {X 85.1496,Y 70.1495,Z 113,A 35.2331,B 24.9325,C -1.8974,E1 25.123,E2 410.4722} C_DIS
LIN {X 82.5998,Y 73.1356,Z 113,A 38.1351,B 24.9294,C -1.9403,E1 25.1175,E2 407.4819} C_DIS
LIN {X 79.4962,Y 76.4955,Z 113,A 39.6909,B 24.9317,C -1.9093,E1 25.1147,E2 406.006} C_DIS
LIN {X 77.4872,Y 78.5297,Z 113,A 41.2894,B 24.9311,C -1.9175,E1 25.1115,E2 404.395} C_DIS
LIN {X 74.6214,Y 81.2578,Z 113,A 43.2162,B 24.9311,C -1.9162,E1 25.1076,E2 402.4793} C_DIS
LIN {X 72.4095,Y 83.2352,Z 113,A 44.8369,B 24.9307,C -1.9227,E1 25.1042,E2 400.8495} C_DIS
LIN {X 69.2772,Y 85.8598,Z 113,A 47.0547,B 24.9301,C -1.9309,E1 25.0994,E2 398.6208} C_DIS
LIN {X 65.6138,Y 88.6922,Z 113,A 49.4454,B 24.9298,C -1.9346,E1 25.094,E2 396.23} C_DIS
LIN {X 62.6417,Y 90.815,Z 113,A 51.9327,B 24.9277,C -1.9636,E1 25.0882,E2 393.6827} C_DIS
LIN {X 58.8396,Y 93.3236,Z 113,A 53.4373,B 24.9302,C -1.9299,E1 25.0849,E2 392.2628} C_DIS
LIN {X 55.0979,Y 95.5795,Z 113,A 56.3864,B 24.9278,C -1.9626,E1 25.0776,E2 389.2452} C_DIS
LIN {X 51.7182,Y 97.4502,Z 113,A 57.8359,B 24.9293,C -1.9413,E1 25.0742,E2 387.8502} C_DIS
LIN {X 48.9787,Y 98.8548,Z 113,A 60.1317,B 24.927,C -1.9734,E1 25.0682,E2 385.4847} C_DIS
LIN {X 44.8826,Y 100.7818,Z 113,A 61.5794,B 24.9296,C -1.9373,E1 25.0648,E2 384.126} C_DIS
LIN {X 41.2424,Y 102.325,Z 113,A 63.9624,B 24.9285,C -1.9535,E1 25.0586,E2 381.7102} C_DIS
LIN {X 34.327,Y 104.8475,Z 113,A 67.4679,B 24.9292,C -1.9434,E1 25.0494,E2 378.2357} C_DIS
LIN {X 31.8975,Y 105.6126,Z 113,A 69.2723,B 24.9276,C -1.9648,E1 25.0445,E2 376.384} C_DIS
LIN {X 28.1383,Y 106.6764,Z 113,A 71.3834,B 24.9273,C -1.9696,E1 25.0388,E2 374.2648} C_DIS
LIN {X 24.3258,Y 107.6091,Z 113,A 73.1693,B 24.928,C -1.96,E1 25.034,E2 372.5041} C_DIS
LIN {X 20.8692,Y 108.3313,Z 113,A 74.8782,B 24.9283,C -1.9556,E1 25.0293,E2 370.8077} C_DIS
LIN {X 17.3115,Y 108.9574,Z 113,A 76.8171,B 24.9281,C -1.9589,E1 25.024,E2 368.8631} C_DIS
LIN {X 14.058,Y 109.4238,Z 113,A 78.4626,B 24.9282,C -1.9567,E1 25.0194,E2 367.2241} C_DIS
LIN {X 10.5227,Y 109.8208,Z 113,A 80.4028,B 24.9279,C -1.9608,E1 25.014,E2 365.2754} C_DIS
LIN {X 6.5743,Y 110.1281,Z 113,A 82.4362,B 24.9279,C -1.9599,E1 25.0084,E2 363.2451} C_DIS
LIN {X 3.3077,Y 110.2735,Z 113,A 84.1511,B 24.9279,C -1.9605,E1 25.0036,E2 361.5292} C_DIS
LIN {X -0.5853,Y 110.3216,Z 113,A 86.0773,B 24.9283,C -1.9562,E1 24.9982,E2 359.6135} C_DIS
LIN {X -3.7266,Y 110.2607,Z 113,A 87.6916,B 24.9283,C -1.955,E1 24.9937,E2 358.0018} C_DIS
LIN {X -7.3842,Y 110.0757,Z 113,A 89.6225,B 24.9283,C -1.9554,E1 24.9883,E2 356.0692} C_DIS
LIN {X -10.9316,Y 109.7816,Z 113,A 91.6012,B 24.928,C -1.9598,E1 24.9828,E2 354.0791} C_DIS
LIN {X -14.8267,Y 109.3242,Z 113,A 93.6195,B 24.9281,C -1.9578,E1 24.9772,E2 352.064} C_DIS
LIN {X -18.1277,Y 108.8236,Z 113,A 95.8489,B 24.9267,C -1.9769,E1 24.971,E2 349.7873} C_DIS
LIN {X -22.1907,Y 108.0683,Z 113,A 97.4282,B 24.9286,C -1.952,E1 24.9668,E2 348.2653} C_DIS
LIN {X -25.9963,Y 107.2166,Z 113,A 100.3979,B 24.9259,C -1.9886,E1 24.9585,E2 345.2046} C_DIS
LIN {X -31.4907,Y 105.7333,Z 113,A 102.4261,B 24.9289,C -1.9476,E1 24.9533,E2 343.2706} C_DIS
LIN {X -37.7439,Y 103.6658,Z 113,A 105.8199,B 24.9293,C -1.9423,E1 24.9444,E2 339.8829} C_DIS
LIN {X -40.7275,Y 102.5311,Z 113,A 108.1175,B 24.9276,C -1.9657,E1 24.9382,E2 337.5246} C_DIS
LIN {X -44.7211,Y 100.8546,Z 113,A 109.9095,B 24.9291,C -1.944,E1 24.9338,E2 335.7801} C_DIS
LIN {X -48.1599,Y 99.2572,Z 113,A 111.845,B 24.9295,C -1.9396,E1 24.9289,E2 333.8501} C_DIS
LIN {X -52.0404,Y 97.2799,Z 113,A 114.0857,B 24.9298,C -1.9349,E1 24.9233,E2 331.6143} C_DIS
LIN {X -55.3375,Y 95.4418,Z 113,A 116.0671,B 24.93,C -1.9323,E1 24.9185,E2 329.6333} C_DIS
LIN {X -58.7468,Y 93.3816,Z 113,A 118.0684,B 24.9305,C -1.9258,E1 24.9138,E2 327.6414} C_DIS
LIN {X -65.2299,Y 88.9733,Z 113,A 122.1494,B 24.931,C -1.9179,E1 24.9045,E2 323.5652} C_DIS
LIN {X -70.0561,Y 85.2272,Z 113,A 125.2113,B 24.9319,C -1.9066,E1 24.8978,E2 320.5188} C_DIS
LIN {X -73.7835,Y 82.0198,Z 113,A 127.8353,B 24.9321,C -1.9035,E1 24.8923,E2 317.8919} C_DIS
LIN {X -77.0779,Y 78.9323,Z 113,A 130.4154,B 24.9318,C -1.9071,E1 24.887,E2 315.2926} C_DIS
LIN {X -80.6088,Y 75.3228,Z 113,A 133.2004,B 24.9318,C -1.907,E1 24.8816,E2 312.4959} C_DIS
LIN {X -84.2593,Y 71.2153,Z 113,A 136.3844,B 24.9314,C -1.9125,E1 24.8758,E2 309.2842} C_DIS
LIN {X -87.0092,Y 67.83,Z 113,A 138.7305,B 24.9316,C -1.9096,E1 24.8717,E2 306.934} C_DIS
LIN {X -89.7169,Y 64.2035,Z 113,A 140.3011,B 24.9342,C -1.8728,E1 24.8693,E2 305.4433} C_DIS
LIN {X -91.379,Y 61.8147,Z 113,A 142.6647,B 24.9322,C -1.9017,E1 24.8655,E2 302.9992} C_DIS
LIN {X -94.0086,Y 57.7395,Z 113,A 144.3052,B 24.9351,C -1.8604,E1 24.8632,E2 301.4487} C_DIS
LIN {X -95.5634,Y 55.1258,Z 113,A 146.097,B 24.9349,C -1.864,E1 24.8606,E2 299.6391} C_DIS
LIN {X -97.4601,Y 51.6994,Z 113,A 148.3733,B 24.9346,C -1.8674,E1 24.8576,E2 297.3427} C_DIS
LIN {X -99.5246,Y 47.6034,Z 113,A 150.4328,B 24.936,C -1.8478,E1 24.8551,E2 295.3187} C_DIS
LIN {X -100.9288,Y 44.5512,Z 113,A 152.0901,B 24.9366,C -1.8391,E1 24.8532,E2 293.673} C_DIS
LIN {X -102.0321,Y 41.9619,Z 113,A 154.3434,B 24.9348,C -1.8651,E1 24.8507,E2 291.3453} C_DIS
LIN {X -103.5781,Y 37.9841,Z 113,A 155.9548,B 24.9369,C -1.8349,E1 24.8492,E2 289.7967} C_DIS
LIN {X -104.7439,Y 34.6453,Z 113,A 158.3129,B 24.9359,C -1.8492,E1 24.8471,E2 287.3912} C_DIS
LIN {X -105.859,Y 31.0669,Z 113,A 159.6598,B 24.9379,C -1.82,E1 24.846,E2 286.106} C_DIS
LIN {X -107.4833,Y 24.8704,Z 113,A 163.0806,B 24.9384,C -1.8129,E1 24.8437,E2 282.6822} C_DIS
LIN {X -108.224,Y 21.4263,Z 113,A 165.1504,B 24.9382,C -1.8162,E1 24.8425,E2 280.5923} C_DIS
LIN {X -109.1118,Y 16.3125,Z 113,A 167.7212,B 24.9391,C -1.8027,E1 24.8413,E2 278.0384} C_DIS
LIN {X -109.5766,Y 12.8122,Z 113,A 169.5101,B 24.9396,C -1.7951,E1 24.8407,E2 276.257} C_DIS
LIN {X -110.0925,Y 7.1363,Z 113,A 172.4145,B 24.9404,C -1.7833,E1 24.8401,E2 273.3633} C_DIS
LIN {X -110.3066,Y 1.9131,Z 113,A 175.1029,B 24.9411,C -1.7735,E1 24.8398,E2 270.6821} C_DIS
LIN {X -110.3178,Y -1.2204,Z 113,A 177.3452,B 24.9398,C -1.7918,E1 24.8398,E2 268.3826} C_DIS
LIN {X -110.2185,Y -4.8046,Z 113,A 179.0871,B 24.9405,C -1.7811,E1 24.8401,E2 266.6556} C_DIS
LIN {X -110.033,Y -8.0154,Z 113,A -179.7105,B 24.9421,C -1.7578,E1 24.8403,E2 265.5018} C_DIS
LIN {X -109.6487,Y -12.1967,Z 113,A -176.8738,B 24.9409,C -1.776,E1 24.8411,E2 262.6045} C_DIS
LIN {X -109.1742,Y -15.8844,Z 113,A -174.8306,B 24.9409,C -1.7743,E1 24.8419,E2 260.5533} C_DIS
LIN {X -108.4825,Y -20.076,Z 113,A -173.3332,B 24.9433,C -1.7399,E1 24.8427,E2 259.129} C_DIS
LIN {X -107.4725,Y -24.917,Z 113,A -170.3504,B 24.9427,C -1.7479,E1 24.8444,E2 256.1096} C_DIS
LIN {X -106.6705,Y -28.16,Z 113,A -168.4713,B 24.9427,C -1.7481,E1 24.8458,E2 254.2192} C_DIS
LIN {X -105.7884,Y -31.305,Z 113,A -167.5342,B 24.945,C -1.7136,E1 24.8465,E2 253.3588} C_DIS
LIN {X -105.0297,Y -33.7637,Z 113,A -165.8622,B 24.9444,C -1.7225,E1 24.8479,E2 251.6561} C_DIS
LIN {X -104.0637,Y -36.6325,Z 113,A -164.2968,B 24.9447,C -1.7175,E1 24.8493,E2 250.0936} C_DIS
LIN {X -102.8715,Y -39.861,Z 113,A -162.4083,B 24.9448,C -1.7161,E1 24.8512,E2 248.1977} C_DIS
LIN {X -101.4129,Y -43.44,Z 113,A -160.5239,B 24.9455,C -1.7055,E1 24.8532,E2 246.3282} C_DIS
LIN {X -99.8634,Y -46.8889,Z 113,A -158.3514,B 24.9453,C -1.708,E1 24.8557,E2 244.1378} C_DIS
LIN {X -98.1054,Y -50.4638,Z 113,A -156.0794,B 24.9452,C -1.7102,E1 24.8586,E2 241.8485} C_DIS
LIN {X -95.831,Y -54.6602,Z 113,A -153.8445,B 24.9462,C -1.6939,E1 24.8616,E2 239.6407} C_DIS
LIN {X -93.912,Y -57.8978,Z 113,A -151.1521,B 24.9447,C -1.7177,E1 24.8657,E2 236.8778} C_DIS
LIN {X -91.3217,Y -61.8994,Z 113,A -149.4088,B 24.947,C -1.6825,E1 24.8682,E2 235.2097} C_DIS
LIN {X -89.0249,Y -65.1594,Z 113,A -146.8762,B 24.9461,C -1.6955,E1 24.8724,E2 232.6338} C_DIS
LIN {X -86.817,Y -68.0748,Z 113,A -145.3849,B 24.9474,C -1.6747,E1 24.8749,E2 231.1848} C_DIS
LIN {X -84.808,Y -70.5606,Z 113,A -143.7478,B 24.9477,C -1.6699,E1 24.8778,E2 229.5516} C_DIS
Enddeposition()
END
